LIN {X 0,Y 113.394,Z 388.758,A -85,B 0,C 180,E1 -26470.714,E2 -26470.714} C_VEL
LIN {X 0,Y 109.1,Z 389.64,A -85,B 0,C 180,E1 -26474.93,E2 -26474.93} C_VEL
LIN {X 0,Y 104.868,Z 389.896,A -85,B 0,C 180,E1 -26480.244,E2 -26480.244} C_VEL
LIN {X 0,Y 101.559,Z 389.287,A -85,B 0,C 180,E1 -26485.896,E2 -26485.896} C_VEL
LIN {X 0,Y 99.232,Z 387.805,A -85,B 0,C 180,E1 -26491.803,E2 -26491.803} C_VEL
LIN {X 0,Y 97.668,Z 384.272,A -85,B 0,C 180,E1 -26500.36,E2 -26500.36} C_VEL
LIN {X 0,Y 97.717,Z 379.628,A -85,B 0,C 180,E1 -26507.919,E2 -26507.919} C_VEL
LIN {X 0,Y 98.543,Z 374.936,A -85,B 0,C 180,E1 -26513.645,E2 -26513.645} C_VEL
LIN {X 0,Y 99.92,Z 369.096,A -85,B 0,C 180,E1 -26519.29,E2 -26519.29} C_VEL
LIN {X 0,Y 102.004,Z 361.819,A -85,B 0,C 180,E1 -26524.852,E2 -26524.852} C_VEL
LIN {X 0,Y 104.986,Z 352.316,A -85,B 0,C 180,E1 -26530.446,E2 -26530.446} C_VEL
LIN {X 0,Y 108.19,Z 342.332,A -85,B 0,C 180,E1 -26534.94,E2 -26534.94} C_VEL
LIN {X 0,Y 111.403,Z 331.682,A -85,B 0,C 180,E1 -26538.631,E2 -26538.631} C_VEL
LIN {X 0,Y 114.734,Z 319.038,A -85,B 0,C 180,E1 -26541.907,E2 -26541.907} C_VEL
LIN {X 0,Y 117.58,Z 306.377,A -85,B 0,C 180,E1 -26544.3,E2 -26544.3} C_VEL
LIN {X 0,Y 119.75,Z 292.877,A -85,B 0,C 180,E1 -26546.101,E2 -26546.101} C_VEL
LIN {X 0,Y 121.436,Z 279.148,A -85,B 0,C 180,E1 -26547.229,E2 -26547.229} C_VEL
LIN {X 0,Y 124.892,Z 239.128,A -85,B 0,C 180,E1 -26549.691,E2 -26549.691} C_VEL
LIN {X 0,Y 118.851,Z 223.709,A -85,B 0,C 180,E1 -26552.831,E2 -26552.831} C_VEL
LIN {X 0,Y 112.352,Z 209.651,A -85,B 0,C 180,E1 -26556.477,E2 -26556.477} C_VEL
LIN {X 0,Y 105.334,Z 198.402,A -85,B 0,C 180,E1 -26560.607,E2 -26560.607} C_VEL
LIN {X 0,Y 103.347,Z 195.213,A -85,B 0,C 180,E1 -26561.916,E2 -26561.916} C_VEL
LIN {X 0,Y 101.464,Z 192.565,A -85,B 0,C 180,E1 -26563.185,E2 -26563.185} C_VEL
LIN {X 0,Y 101.019,Z 190.903,A -85,B 0,C 180,E1 -26563.693,E2 -26563.693} C_VEL
LIN {X 0,Y 100.77,Z 190.929,A -85,B 0,C 180,E1 -26570.409,E2 -26570.409} C_VEL
LIN {X 0,Y 100.714,Z 190.936,A -85,B 0,C 180,E1 -26574.889,E2 -26574.889} C_VEL
LIN {X 0,Y 100.681,Z 190.926,A -85,B 0,C 180,E1 -26583.11,E2 -26583.11} C_VEL
LIN {X 0,Y 100.629,Z 190.942,A -85,B 0,C 180,E1 -26589.806,E2 -26589.806} C_VEL
LIN {X 0,Y 100.634,Z 190.932,A -85,B 0,C 180,E1 -26595.706,E2 -26595.706} C_VEL
LIN {X 0,Y 100.619,Z 190.949,A -85,B 0,C 180,E1 -26601.053,E2 -26601.053} C_VEL
LIN {X 0,Y 100.682,Z 190.91,A -85,B 0,C 180,E1 -26606.893,E2 -26606.893} C_VEL
LIN {X 0,Y 100.723,Z 190.936,A -85,B 0,C 180,E1 -26615.252,E2 -26615.252} C_VEL
LIN {X 0,Y 100.77,Z 190.902,A -85,B 0,C 180,E1 -26619.593,E2 -26619.593} C_VEL
LIN {X 0,Y 101.113,Z 190.885,A -85,B 0,C 180,E1 -26627.966,E2 -26627.966} C_VEL
LIN {X 0,Y 101.216,Z 190.86,A -85,B 0,C 180,E1 -26632.019,E2 -26632.019} C_VEL
LIN {X 0,Y 101.822,Z 190.796,A -85,B 0,C 180,E1 -26640.002,E2 -26640.002} C_VEL
LIN {X 0,Y 101.217,Z 190.855,A -85,B 0,C 180,E1 -26647.984,E2 -26647.984} C_VEL
LIN {X 0,Y 101.05,Z 190.897,A -85,B 0,C 180,E1 -26653.17,E2 -26653.17} C_VEL
LIN {X 0,Y 100.772,Z 190.934,A -85,B 0,C 180,E1 -26660.41,E2 -26660.41} C_VEL
LIN {X 0,Y 100.701,Z 190.933,A -85,B 0,C 180,E1 -26664.868,E2 -26664.868} C_VEL
LIN {X 0,Y 100.636,Z 190.954,A -85,B 0,C 180,E1 -26669.698,E2 -26669.698} C_VEL
LIN {X 0,Y 101.603,Z 193.649,A -85,B 0,C 180,E1 -26670.531,E2 -26670.531} C_VEL
LIN {X 0,Y 103.52,Z 196.141,A -85,B 0,C 180,E1 -26671.784,E2 -26671.784} C_VEL
LIN {X 0,Y 109.673,Z 206.47,A -85,B 0,C 180,E1 -26675.645,E2 -26675.645} C_VEL
LIN {X 0,Y 115.294,Z 217.308,A -85,B 0,C 180,E1 -26678.881,E2 -26678.881} C_VEL
LIN {X 0,Y 120.773,Z 232.647,A -85,B 0,C 180,E1 -26682.073,E2 -26682.073} C_VEL
LIN {X 0,Y 124.213,Z 244.441,A -85,B 0,C 180,E1 -26684.089,E2 -26684.089} C_VEL
LIN {X 0,Y 124.314,Z 249.248,A -85,B 0,C 180,E1 -26684.526,E2 -26684.526} C_VEL
LIN {X 0,Y 120.506,Z 292.686,A -85,B 0,C 180,E1 -26687.314,E2 -26687.314} C_VEL
LIN {X 0,Y 118.54,Z 305.908,A -85,B 0,C 180,E1 -26688.732,E2 -26688.732} C_VEL
LIN {X 0,Y 116.204,Z 317.72,A -85,B 0,C 180,E1 -26690.577,E2 -26690.577} C_VEL
LIN {X 0,Y 113.003,Z 330.055,A -85,B 0,C 180,E1 -26693.23,E2 -26693.23} C_VEL
LIN {X 0,Y 109.597,Z 341.808,A -85,B 0,C 180,E1 -26696.664,E2 -26696.664} C_VEL
LIN {X 0,Y 106.566,Z 351.426,A -85,B 0,C 180,E1 -26700.355,E2 -26700.355} C_VEL
LIN {X 0,Y 103.695,Z 360.644,A -85,B 0,C 180,E1 -26704.938,E2 -26704.938} C_VEL
LIN {X 0,Y 101.014,Z 369.603,A -85,B 0,C 180,E1 -26710.702,E2 -26710.702} C_VEL
LIN {X 0,Y 99.294,Z 376.773,A -85,B 0,C 180,E1 -26716.701,E2 -26716.701} C_VEL
LIN {X 0,Y 98.557,Z 381.59,A -85,B 0,C 180,E1 -26721.8,E2 -26721.8} C_VEL
LIN {X 0,Y 98.327,Z 386.191,A -85,B 0,C 180,E1 -26727.951,E2 -26727.951} C_VEL
LIN {X 0,Y 98.286,Z 388.572,A -85,B 0,C 180,E1 -26732.048,E2 -26732.048} C_VEL
LIN {X 0,Y 98.411,Z 391.267,A -85,B 0,C 180,E1 -26738.211,E2 -26738.211} C_VEL
LIN {X 0,Y 100,Z 393.408,A -85,B 0,C 180,E1 -26746.326,E2 -26746.326} C_VEL
LIN {X 0,Y 103.424,Z 394.112,A -85,B 0,C 180,E1 -26754.061,E2 -26754.061} C_VEL
LIN {X 0,Y 108.893,Z 393.383,A -85,B 0,C 180,E1 -26761.085,E2 -26761.085} C_VEL
LIN {X 0,Y 115.931,Z 391.168,A -85,B 0,C 180,E1 -26767.316,E2 -26767.316} C_VEL
LIN {X 0,Y 124.081,Z 387.478,A -85,B 0,C 180,E1 -26772.818,E2 -26772.818} C_VEL
LIN {X 0,Y 131.12,Z 383.572,A -85,B 0,C 180,E1 -26776.351,E2 -26776.351} C_VEL
LIN {X 0,Y 138.522,Z 378.707,A -85,B 0,C 180,E1 -26779.554,E2 -26779.554} C_VEL
LIN {X 0,Y 146.531,Z 372.647,A -85,B 0,C 180,E1 -26782.313,E2 -26782.313} C_VEL
LIN {X 0,Y 154.92,Z 365.206,A -85,B 0,C 180,E1 -26784.742,E2 -26784.742} C_VEL
LIN {X 0,Y 163.564,Z 356.027,A -85,B 0,C 180,E1 -26786.914,E2 -26786.914} C_VEL
LIN {X 0,Y 170.963,Z 346.797,A -85,B 0,C 180,E1 -26788.537,E2 -26788.537} C_VEL
LIN {X 0,Y 178.613,Z 335.405,A -85,B 0,C 180,E1 -26789.955,E2 -26789.955} C_VEL
LIN {X 0,Y 184.843,Z 323.877,A -85,B 0,C 180,E1 -26790.983,E2 -26790.983} C_VEL
LIN {X 0,Y 190.498,Z 310.611,A -85,B 0,C 180,E1 -26791.832,E2 -26791.832} C_VEL
LIN {X 0,Y 194.101,Z 299.386,A -85,B 0,C 180,E1 -26792.328,E2 -26792.328} C_VEL
LIN {X 0,Y 194.458,Z 297.623,A -85,B 0,C 180,E1 -26792.68,E2 -26792.68} C_VEL
LIN {X 0,Y 194.529,Z 296.426,A -85,B 0,C 180,E1 -26793.471,E2 -26793.471} C_VEL
LIN {X 0,Y 194.251,Z 296.2,A -85,B 0,C 180,E1 -26794.794,E2 -26794.794} C_VEL
LIN {X 0,Y 193.484,Z 297.975,A -85,B 0,C 180,E1 -26798.13,E2 -26798.13} C_VEL
LIN {X 0,Y 193.518,Z 298.009,A -85,B 0,C 180,E1 -26798.613,E2 -26798.613} C_VEL
LIN {X 0,Y 193.642,Z 298.314,A -85,B 0,C 180,E1 -26799.96,E2 -26799.96} C_VEL
LIN {X 0,Y 189.131,Z 311.645,A -85,B 0,C 180,E1 -26800.643,E2 -26800.643} C_VEL
LIN {X 0,Y 183.324,Z 324.478,A -85,B 0,C 180,E1 -26801.574,E2 -26801.574} C_VEL
LIN {X 0,Y 176.612,Z 336.059,A -85,B 0,C 180,E1 -26802.751,E2 -26802.751} C_VEL
LIN {X 0,Y 168.731,Z 347.161,A -85,B 0,C 180,E1 -26804.278,E2 -26804.278} C_VEL
LIN {X 0,Y 161.82,Z 355.239,A -85,B 0,C 180,E1 -26805.75,E2 -26805.75} C_VEL
LIN {X 0,Y 153.509,Z 363.475,A -85,B 0,C 180,E1 -26807.76,E2 -26807.76} C_VEL
LIN {X 0,Y 143.868,Z 371.395,A -85,B 0,C 180,E1 -26810.488,E2 -26810.488} C_VEL
LIN {X 0,Y 134.326,Z 377.914,A -85,B 0,C 180,E1 -26813.753,E2 -26813.753} C_VEL
LIN {X 0,Y 126.685,Z 382.18,A -85,B 0,C 180,E1 -26816.91,E2 -26816.91} C_VEL
LIN {X 0,Y 119.479,Z 385.482,A -85,B 0,C 180,E1 -26820.549,E2 -26820.549} C_VEL
LIN {X 0,Y 112.816,Z 387.875,A -85,B 0,C 180,E1 -26824.647,E2 -26824.647} C_VEL
LIN {X 0,Y 106.817,Z 389.413,A -85,B 0,C 180,E1 -26829.287,E2 -26829.287} C_VEL
LIN {X 0,Y 100.124,Z 390.135,A -85,B 0,C 180,E1 -26836.304,E2 -26836.304} C_VEL
LIN {X 0,Y 96.622,Z 389.783,A -85,B 0,C 180,E1 -26841.325,E2 -26841.325} C_VEL
LIN {X 0,Y 93.832,Z 388.808,A -85,B 0,C 180,E1 -26846.703,E2 -26846.703} C_VEL
LIN {X 0,Y 91.202,Z 385.997,A -85,B 0,C 180,E1 -26855.301,E2 -26855.301} C_VEL
LIN {X 0,Y 90.512,Z 383.048,A -85,B 0,C 180,E1 -26861.591,E2 -26861.591} C_VEL
LIN {X 0,Y 90.639,Z 379.163,A -85,B 0,C 180,E1 -26867.946,E2 -26867.946} C_VEL
LIN {X 0,Y 91.636,Z 373.852,A -85,B 0,C 180,E1 -26874.658,E2 -26874.658} C_VEL
LIN {X 0,Y 93.142,Z 367.817,A -85,B 0,C 180,E1 -26880.631,E2 -26880.631} C_VEL
LIN {X 0,Y 95.227,Z 360.904,A -85,B 0,C 180,E1 -26886.053,E2 -26886.053} C_VEL
LIN {X 0,Y 98.32,Z 351.51,A -85,B 0,C 180,E1 -26891.777,E2 -26891.777} C_VEL
LIN {X 0,Y 101.719,Z 341.4,A -85,B 0,C 180,E1 -26896.485,E2 -26896.485} C_VEL
LIN {X 0,Y 105.411,Z 329.532,A -85,B 0,C 180,E1 -26900.608,E2 -26900.608} C_VEL
LIN {X 0,Y 108.633,Z 317.539,A -85,B 0,C 180,E1 -26903.733,E2 -26903.733} C_VEL
LIN {X 0,Y 111.595,Z 304.439,A -85,B 0,C 180,E1 -26906.164,E2 -26906.164} C_VEL
LIN {X 0,Y 113.783,Z 291.045,A -85,B 0,C 180,E1 -26907.922,E2 -26907.922} C_VEL
LIN {X 0,Y 115.568,Z 275.498,A -85,B 0,C 180,E1 -26909.114,E2 -26909.114} C_VEL
LIN {X 0,Y 118.609,Z 240.464,A -85,B 0,C 180,E1 -26911.383,E2 -26911.383} C_VEL
LIN {X 0,Y 113.185,Z 226.664,A -85,B 0,C 180,E1 -26914.475,E2 -26914.475} C_VEL
LIN {X 0,Y 107.453,Z 213.945,A -85,B 0,C 180,E1 -26917.984,E2 -26917.984} C_VEL
LIN {X 0,Y 99.311,Z 200.557,A -85,B 0,C 180,E1 -26923.337,E2 -26923.337} C_VEL
LIN {X 0,Y 97,Z 197.039,A -85,B 0,C 180,E1 -26925.059,E2 -26925.059} C_VEL
LIN {X 0,Y 94.472,Z 194.146,A -85,B 0,C 180,E1 -26926.939,E2 -26926.939} C_VEL
LIN {X 0,Y 93.716,Z 191.812,A -85,B 0,C 180,E1 -26927.879,E2 -26927.879} C_VEL
LIN {X 0,Y 93.628,Z 191.82,A -85,B 0,C 180,E1 -26935.747,E2 -26935.747} C_VEL
LIN {X 0,Y 93.579,Z 191.817,A -85,B 0,C 180,E1 -26944.301,E2 -26944.301} C_VEL
LIN {X 0,Y 93.521,Z 191.808,A -85,B 0,C 180,E1 -26952.558,E2 -26952.558} C_VEL
LIN {X 0,Y 93.527,Z 191.833,A -85,B 0,C 180,E1 -26958.715,E2 -26958.715} C_VEL
LIN {X 0,Y 93.579,Z 191.795,A -85,B 0,C 180,E1 -26965.703,E2 -26965.703} C_VEL
LIN {X 0,Y 93.629,Z 191.822,A -85,B 0,C 180,E1 -26974.256,E2 -26974.256} C_VEL
LIN {X 0,Y 93.64,Z 191.804,A -85,B 0,C 180,E1 -26977.961,E2 -26977.961} C_VEL
LIN {X 0,Y 94.014,Z 191.768,A -85,B 0,C 180,E1 -26987.042,E2 -26987.042} C_VEL
LIN {X 0,Y 94.128,Z 191.746,A -85,B 0,C 180,E1 -26991.414,E2 -26991.414} C_VEL
LIN {X 0,Y 94.751,Z 191.677,A -85,B 0,C 180,E1 -27000.002,E2 -27000.002} C_VEL
LIN {X 0,Y 94.129,Z 191.741,A -85,B 0,C 180,E1 -27008.59,E2 -27008.59} C_VEL
LIN {X 0,Y 93.958,Z 191.779,A -85,B 0,C 180,E1 -27013.495,E2 -27013.495} C_VEL
LIN {X 0,Y 93.635,Z 191.821,A -85,B 0,C 180,E1 -27022.044,E2 -27022.044} C_VEL
LIN {X 0,Y 93.615,Z 191.818,A -85,B 0,C 180,E1 -27025.727,E2 -27025.727} C_VEL
LIN {X 0,Y 94.495,Z 194.57,A -85,B 0,C 180,E1 -27026.654,E2 -27026.654} C_VEL
LIN {X 0,Y 96.723,Z 197.337,A -85,B 0,C 180,E1 -27028.333,E2 -27028.333} C_VEL
LIN {X 0,Y 100.215,Z 202.921,A -85,B 0,C 180,E1 -27030.943,E2 -27030.943} C_VEL
LIN {X 0,Y 105.187,Z 211.401,A -85,B 0,C 180,E1 -27034.281,E2 -27034.281} C_VEL
LIN {X 0,Y 110.057,Z 220.958,A -85,B 0,C 180,E1 -27037.296,E2 -27037.296} C_VEL
LIN {X 0,Y 114.862,Z 234.875,A -85,B 0,C 180,E1 -27040.409,E2 -27040.409} C_VEL
LIN {X 0,Y 118.188,Z 246.008,A -85,B 0,C 180,E1 -27042.492,E2 -27042.492} C_VEL
LIN {X 0,Y 118.164,Z 250.07,A -85,B 0,C 180,E1 -27042.85,E2 -27042.85} C_VEL
LIN {X 0,Y 114.327,Z 291.924,A -85,B 0,C 180,E1 -27045.633,E2 -27045.633} C_VEL
LIN {X 0,Y 112.15,Z 305.956,A -85,B 0,C 180,E1 -27047.193,E2 -27047.193} C_VEL
LIN {X 0,Y 109.847,Z 317.152,A -85,B 0,C 180,E1 -27049.02,E2 -27049.02} C_VEL
LIN {X 0,Y 106.496,Z 329.581,A -85,B 0,C 180,E1 -27051.78,E2 -27051.78} C_VEL
LIN {X 0,Y 103.154,Z 340.625,A -85,B 0,C 180,E1 -27055.122,E2 -27055.122} C_VEL
LIN {X 0,Y 99.746,Z 351.044,A -85,B 0,C 180,E1 -27059.281,E2 -27059.281} C_VEL
LIN {X 0,Y 96.725,Z 360.293,A -85,B 0,C 180,E1 -27064.154,E2 -27064.154} C_VEL
LIN {X 0,Y 94.34,Z 367.912,A -85,B 0,C 180,E1 -27069.276,E2 -27069.276} C_VEL
LIN {X 0,Y 92.395,Z 375.362,A -85,B 0,C 180,E1 -27075.687,E2 -27075.687} C_VEL
LIN {X 0,Y 91.548,Z 380.394,A -85,B 0,C 180,E1 -27081.168,E2 -27081.168} C_VEL
LIN {X 0,Y 91.27,Z 385.199,A -85,B 0,C 180,E1 -27087.793,E2 -27087.793} C_VEL
LIN {X 0,Y 91.254,Z 387.713,A -85,B 0,C 180,E1 -27092.206,E2 -27092.206} C_VEL
LIN {X 0,Y 91.421,Z 390.547,A -85,B 0,C 180,E1 -27098.843,E2 -27098.843} C_VEL
LIN {X 0,Y 93.206,Z 392.966,A -85,B 0,C 180,E1 -27107.553,E2 -27107.553} C_VEL
LIN {X 0,Y 96.974,Z 393.865,A -85,B 0,C 180,E1 -27115.774,E2 -27115.774} C_VEL
LIN {X 0,Y 102.86,Z 393.366,A -85,B 0,C 180,E1 -27123.133,E2 -27123.133} C_VEL
LIN {X 0,Y 110.375,Z 391.434,A -85,B 0,C 180,E1 -27129.548,E2 -27129.548} C_VEL
LIN {X 0,Y 118.992,Z 387.979,A -85,B 0,C 180,E1 -27135.132,E2 -27135.132} C_VEL
LIN {X 0,Y 126.363,Z 384.345,A -85,B 0,C 180,E1 -27138.661,E2 -27138.661} C_VEL
LIN {X 0,Y 134.082,Z 379.734,A -85,B 0,C 180,E1 -27141.833,E2 -27141.833} C_VEL
LIN {X 0,Y 142.358,Z 373.954,A -85,B 0,C 180,E1 -27144.544,E2 -27144.544} C_VEL
LIN {X 0,Y 152.488,Z 365.565,A -85,B 0,C 180,E1 -27147.257,E2 -27147.257} C_VEL
LIN {X 0,Y 161.404,Z 356.639,A -85,B 0,C 180,E1 -27149.311,E2 -27149.311} C_VEL
LIN {X 0,Y 169.808,Z 346.514,A -85,B 0,C 180,E1 -27150.962,E2 -27150.962} C_VEL
LIN {X 0,Y 176.853,Z 336.34,A -85,B 0,C 180,E1 -27152.15,E2 -27152.15} C_VEL
LIN {X 0,Y 183.235,Z 325.172,A -85,B 0,C 180,E1 -27153.093,E2 -27153.093} C_VEL
LIN {X 0,Y 188.695,Z 313.169,A -85,B 0,C 180,E1 -27153.836,E2 -27153.836} C_VEL
LIN {X 0,Y 193.069,Z 300.628,A -85,B 0,C 180,E1 -27154.372,E2 -27154.372} C_VEL
LIN {X 0,Y 193.419,Z 298.769,A -85,B 0,C 180,E1 -27155.436,E2 -27155.436} C_VEL
LIN {X 0,Y 193.437,Z 298.212,A -85,B 0,C 180,E1 -27156.442,E2 -27156.442} C_VEL
LIN {X 0,Y 193.518,Z 298.009,A -85,B 0,C 180,E1 -27158.613,E2 -27158.613} C_VEL
LIN {X 0,Y 193.353,Z 298.825,A -85,B 0,C 180,E1 -27159.078,E2 -27159.078} C_VEL
LIN {X 0,Y 192.714,Z 301.018,A -85,B 0,C 180,E1 -27159.398,E2 -27159.398} C_VEL
LIN {X 0,Y 191.48,Z 304.858,A -85,B 0,C 180,E1 -27159.451,E2 -27159.451} C_VEL
LIN {X 0,Y 187.404,Z 315.101,A -85,B 0,C 180,E1 -27158.818,E2 -27158.818} C_VEL
LIN {X 0,Y 186.095,Z 317.957,A -85,B 0,C 180,E1 -27158.86,E2 -27158.86} C_VEL
LIN {X 0,Y 180.469,Z 328.902,A -85,B 0,C 180,E1 -27159.694,E2 -27159.694} C_VEL
LIN {X 0,Y 173.566,Z 339.73,A -85,B 0,C 180,E1 -27160.8,E2 -27160.8} C_VEL
LIN {X 0,Y 164.884,Z 350.747,A -85,B 0,C 180,E1 -27162.349,E2 -27162.349} C_VEL
LIN {X 0,Y 155.5,Z 360.522,A -85,B 0,C 180,E1 -27164.265,E2 -27164.265} C_VEL
LIN {X 0,Y 145.774,Z 368.828,A -85,B 0,C 180,E1 -27166.585,E2 -27166.585} C_VEL
LIN {X 0,Y 135.827,Z 375.813,A -85,B 0,C 180,E1 -27169.446,E2 -27169.446} C_VEL
LIN {X 0,Y 127.673,Z 380.498,A -85,B 0,C 180,E1 -27172.23,E2 -27172.23} C_VEL
LIN {X 0,Y 117.527,Z 385.189,A -85,B 0,C 180,E1 -27176.57,E2 -27176.57} C_VEL
LIN {X 0,Y 111.089,Z 387.514,A -85,B 0,C 180,E1 -27179.998,E2 -27179.998} C_VEL
LIN {X 0,Y 105.177,Z 389.089,A -85,B 0,C 180,E1 -27183.83,E2 -27183.83} C_VEL
LIN {X 0,Y 99.463,Z 390.084,A -85,B 0,C 180,E1 -27188.426,E2 -27188.426} C_VEL
LIN {X 0,Y 94.146,Z 390.355,A -85,B 0,C 180,E1 -27193.969,E2 -27193.969} C_VEL
LIN {X 0,Y 89.807,Z 389.757,A -85,B 0,C 180,E1 -27200.106,E2 -27200.106} C_VEL
LIN {X 0,Y 86.517,Z 388.308,A -85,B 0,C 180,E1 -27206.68,E2 -27206.68} C_VEL
LIN {X 0,Y 83.976,Z 385.134,A -85,B 0,C 180,E1 -27215.859,E2 -27215.859} C_VEL
LIN {X 0,Y 83.402,Z 381.981,A -85,B 0,C 180,E1 -27222.384,E2 -27222.384} C_VEL
LIN {X 0,Y 83.684,Z 377.846,A -85,B 0,C 180,E1 -27229.096,E2 -27229.096} C_VEL
LIN {X 0,Y 85.04,Z 371.444,A -85,B 0,C 180,E1 -27237.142,E2 -27237.142} C_VEL
LIN {X 0,Y 87.035,Z 364.395,A -85,B 0,C 180,E1 -27243.881,E2 -27243.881} C_VEL
LIN {X 0,Y 89.785,Z 356.227,A -85,B 0,C 180,E1 -27249.931,E2 -27249.931} C_VEL
LIN {X 0,Y 93.309,Z 346.178,A -85,B 0,C 180,E1 -27255.629,E2 -27255.629} C_VEL
LIN {X 0,Y 96.907,Z 335.656,A -85,B 0,C 180,E1 -27260.083,E2 -27260.083} C_VEL
LIN {X 0,Y 100.743,Z 323.192,A -85,B 0,C 180,E1 -27263.994,E2 -27263.994} C_VEL
LIN {X 0,Y 104.002,Z 310.25,A -85,B 0,C 180,E1 -27266.929,E2 -27266.929} C_VEL
LIN {X 0,Y 106.636,Z 297.298,A -85,B 0,C 180,E1 -27268.992,E2 -27268.992} C_VEL
LIN {X 0,Y 108.567,Z 283.803,A -85,B 0,C 180,E1 -27270.396,E2 -27270.396} C_VEL
LIN {X 0,Y 112.543,Z 242.322,A -85,B 0,C 180,E1 -27273.169,E2 -27273.169} C_VEL
LIN {X 0,Y 107.729,Z 229.872,A -85,B 0,C 180,E1 -27276.197,E2 -27276.197} C_VEL
LIN {X 0,Y 102.538,Z 218.119,A -85,B 0,C 180,E1 -27279.647,E2 -27279.647} C_VEL
LIN {X 0,Y 95.323,Z 205.854,A -85,B 0,C 180,E1 -27284.867,E2 -27284.867} C_VEL
LIN {X 0,Y 92.57,Z 201.95,A -85,B 0,C 180,E1 -27287.034,E2 -27287.034} C_VEL
LIN {X 0,Y 90.181,Z 198.633,A -85,B 0,C 180,E1 -27289.076,E2 -27289.076} C_VEL
LIN {X 0,Y 89.56,Z 197.553,A -85,B 0,C 180,E1 -27289.671,E2 -27289.671} C_VEL
LIN {X 0,Y 87.427,Z 195.251,A -85,B 0,C 180,E1 -27291.611,E2 -27291.611} C_VEL
LIN {X 0,Y 86.559,Z 192.704,A -85,B 0,C 180,E1 -27292.843,E2 -27292.843} C_VEL
LIN {X 0,Y 86.45,Z 192.707,A -85,B 0,C 180,E1 -27299.195,E2 -27299.195} C_VEL
LIN {X 0,Y 86.498,Z 192.707,A -85,B 0,C 180,E1 -27305.662,E2 -27305.662} C_VEL
LIN {X 0,Y 86.446,Z 192.688,A -85,B 0,C 180,E1 -27312.974,E2 -27312.974} C_VEL
LIN {X 0,Y 86.45,Z 192.716,A -85,B 0,C 180,E1 -27319.433,E2 -27319.433} C_VEL
LIN {X 0,Y 86.523,Z 192.674,A -85,B 0,C 180,E1 -27325.35,E2 -27325.35} C_VEL
LIN {X 0,Y 86.553,Z 192.703,A -85,B 0,C 180,E1 -27333.276,E2 -27333.276} C_VEL
LIN {X 0,Y 86.589,Z 192.66,A -85,B 0,C 180,E1 -27341.057,E2 -27341.057} C_VEL
LIN {X 0,Y 86.86,Z 192.655,A -85,B 0,C 180,E1 -27346.153,E2 -27346.153} C_VEL
LIN {X 0,Y 87.023,Z 192.635,A -85,B 0,C 180,E1 -27350.707,E2 -27350.707} C_VEL
LIN {X 0,Y 87.681,Z 192.557,A -85,B 0,C 180,E1 -27360.002,E2 -27360.002} C_VEL
LIN {X 0,Y 87.024,Z 192.63,A -85,B 0,C 180,E1 -27369.297,E2 -27369.297} C_VEL
LIN {X 0,Y 86.86,Z 192.66,A -85,B 0,C 180,E1 -27374.05,E2 -27374.05} C_VEL
LIN {X 0,Y 86.566,Z 192.704,A -85,B 0,C 180,E1 -27380.807,E2 -27380.807} C_VEL
LIN {X 0,Y 87.582,Z 195.517,A -85,B 0,C 180,E1 -27382.097,E2 -27382.097} C_VEL
LIN {X 0,Y 89.771,Z 198.091,A -85,B 0,C 180,E1 -27384.091,E2 -27384.091} C_VEL
LIN {X 0,Y 91.803,Z 201.444,A -85,B 0,C 180,E1 -27385.932,E2 -27385.932} C_VEL
LIN {X 0,Y 95.21,Z 206.474,A -85,B 0,C 180,E1 -27388.656,E2 -27388.656} C_VEL
LIN {X 0,Y 100.921,Z 216.687,A -85,B 0,C 180,E1 -27392.94,E2 -27392.94} C_VEL
LIN {X 0,Y 105.009,Z 225.05,A -85,B 0,C 180,E1 -27395.701,E2 -27395.701} C_VEL
LIN {X 0,Y 109.356,Z 237.939,A -85,B 0,C 180,E1 -27398.765,E2 -27398.765} C_VEL
LIN {X 0,Y 112.259,Z 248.266,A -85,B 0,C 180,E1 -27400.821,E2 -27400.821} C_VEL
LIN {X 0,Y 108.112,Z 292.116,A -85,B 0,C 180,E1 -27403.864,E2 -27403.864} C_VEL
LIN {X 0,Y 105.856,Z 305.968,A -85,B 0,C 180,E1 -27405.471,E2 -27405.471} C_VEL
LIN {X 0,Y 103.061,Z 318.595,A -85,B 0,C 180,E1 -27407.67,E2 -27407.67} C_VEL
LIN {X 0,Y 99.596,Z 330.652,A -85,B 0,C 180,E1 -27410.573,E2 -27410.573} C_VEL
LIN {X 0,Y 96.064,Z 341.656,A -85,B 0,C 180,E1 -27414.177,E2 -27414.177} C_VEL
LIN {X 0,Y 92.968,Z 350.658,A -85,B 0,C 180,E1 -27418.05,E2 -27418.05} C_VEL
LIN {X 0,Y 89.802,Z 359.943,A -85,B 0,C 180,E1 -27423.256,E2 -27423.256} C_VEL
LIN {X 0,Y 87.297,Z 367.557,A -85,B 0,C 180,E1 -27428.759,E2 -27428.759} C_VEL
LIN {X 0,Y 85.285,Z 375,A -85,B 0,C 180,E1 -27435.686,E2 -27435.686} C_VEL
LIN {X 0,Y 84.363,Z 380.936,A -85,B 0,C 180,E1 -27442.821,E2 -27442.821} C_VEL
LIN {X 0,Y 84.298,Z 385.547,A -85,B 0,C 180,E1 -27449.999,E2 -27449.999} C_VEL
LIN {X 0,Y 84.218,Z 387.928,A -85,B 0,C 180,E1 -27454.786,E2 -27454.786} C_VEL
LIN {X 0,Y 85.185,Z 391.316,A -85,B 0,C 180,E1 -27464.329,E2 -27464.329} C_VEL
LIN {X 0,Y 88.239,Z 393.191,A -85,B 0,C 180,E1 -27473.467,E2 -27473.467} C_VEL
LIN {X 0,Y 93.603,Z 393.644,A -85,B 0,C 180,E1 -27481.706,E2 -27481.706} C_VEL
LIN {X 0,Y 100.811,Z 392.649,A -85,B 0,C 180,E1 -27488.859,E2 -27488.859} C_VEL
LIN {X 0,Y 109.89,Z 390.092,A -85,B 0,C 180,E1 -27495.289,E2 -27495.289} C_VEL
LIN {X 0,Y 119.156,Z 386.326,A -85,B 0,C 180,E1 -27500.062,E2 -27500.062} C_VEL
LIN {X 0,Y 127.154,Z 382.278,A -85,B 0,C 180,E1 -27503.265,E2 -27503.265} C_VEL
LIN {X 0,Y 135.522,Z 377.237,A -85,B 0,C 180,E1 -27506.07,E2 -27506.07} C_VEL
LIN {X 0,Y 145.831,Z 369.768,A -85,B 0,C 180,E1 -27508.804,E2 -27508.804} C_VEL
LIN {X 0,Y 154.92,Z 361.834,A -85,B 0,C 180,E1 -27510.84,E2 -27510.84} C_VEL
LIN {X 0,Y 162.647,Z 353.849,A -85,B 0,C 180,E1 -27512.349,E2 -27512.349} C_VEL
LIN {X 0,Y 170.557,Z 344.285,A -85,B 0,C 180,E1 -27513.665,E2 -27513.665} C_VEL
LIN {X 0,Y 177.808,Z 333.657,A -85,B 0,C 180,E1 -27514.706,E2 -27514.706} C_VEL
LIN {X 0,Y 184.344,Z 321.867,A -85,B 0,C 180,E1 -27515.533,E2 -27515.533} C_VEL
LIN {X 0,Y 189.618,Z 309.774,A -85,B 0,C 180,E1 -27516.163,E2 -27516.163} C_VEL
LIN {X 0,Y 190.995,Z 305.941,A -85,B 0,C 180,E1 -27516.299,E2 -27516.299} C_VEL
LIN {X 0,Y 191.309,Z 304.957,A -85,B 0,C 180,E1 -27516.692,E2 -27516.692} C_VEL
LIN {X 0,Y 191.329,Z 304.827,A -85,B 0,C 180,E1 -27517.946,E2 -27517.946} C_VEL
LIN {X 0,Y 191.099,Z 305.504,A -85,B 0,C 180,E1 -27518.17,E2 -27518.17} C_VEL
LIN {X 0,Y 186.095,Z 317.957,A -85,B 0,C 180,E1 -27518.86,E2 -27518.86} C_VEL
LIN {X 0,Y 183.51,Z 323.274,A -85,B 0,C 180,E1 -27518.998,E2 -27518.998} C_VEL
LIN {X 0,Y 178.618,Z 331.896,A -85,B 0,C 180,E1 -27518.77,E2 -27518.77} C_VEL
LIN {X 0,Y 173.123,Z 340.058,A -85,B 0,C 180,E1 -27518.643,E2 -27518.643} C_VEL
LIN {X 0,Y 169.599,Z 344.64,A -85,B 0,C 180,E1 -27518.967,E2 -27518.967} C_VEL
LIN {X 0,Y 160.705,Z 354.796,A -85,B 0,C 180,E1 -27520.419,E2 -27520.419} C_VEL
LIN {X 0,Y 152.901,Z 362.231,A -85,B 0,C 180,E1 -27521.893,E2 -27521.893} C_VEL
LIN {X 0,Y 144.328,Z 369.145,A -85,B 0,C 180,E1 -27523.739,E2 -27523.739} C_VEL
LIN {X 0,Y 134.104,Z 376.055,A -85,B 0,C 180,E1 -27526.356,E2 -27526.356} C_VEL
LIN {X 0,Y 126.201,Z 380.423,A -85,B 0,C 180,E1 -27528.76,E2 -27528.76} C_VEL
LIN {X 0,Y 118.307,Z 384.041,A -85,B 0,C 180,E1 -27531.624,E2 -27531.624} C_VEL
LIN {X 0,Y 108.155,Z 387.669,A -85,B 0,C 180,E1 -27536.273,E2 -27536.273} C_VEL
LIN {X 0,Y 98.463,Z 389.882,A -85,B 0,C 180,E1 -27542.216,E2 -27542.216} C_VEL
LIN {X 0,Y 90.6,Z 390.581,A -85,B 0,C 180,E1 -27548.923,E2 -27548.923} C_VEL
LIN {X 0,Y 86.031,Z 390.296,A -85,B 0,C 180,E1 -27554.184,E2 -27554.184} C_VEL
LIN {X 0,Y 82.271,Z 389.364,A -85,B 0,C 180,E1 -27560.008,E2 -27560.008} C_VEL
LIN {X 0,Y 78.126,Z 386.621,A -85,B 0,C 180,E1 -27569.9,E2 -27569.9} C_VEL
LIN {X 0,Y 76.435,Z 382.436,A -85,B 0,C 180,E1 -27580.06,E2 -27580.06} C_VEL
LIN {X 0,Y 76.462,Z 378.455,A -85,B 0,C 180,E1 -27587.331,E2 -27587.331} C_VEL
LIN {X 0,Y 77.43,Z 373.274,A -85,B 0,C 180,E1 -27594.771,E2 -27594.771} C_VEL
LIN {X 0,Y 79.269,Z 366.397,A -85,B 0,C 180,E1 -27602.444,E2 -27602.444} C_VEL
LIN {X 0,Y 82.318,Z 357.585,A -85,B 0,C 180,E1 -27609.901,E2 -27609.901} C_VEL
LIN {X 0,Y 85.72,Z 348.338,A -85,B 0,C 180,E1 -27615.762,E2 -27615.762} C_VEL
LIN {X 0,Y 89.668,Z 337.386,A -85,B 0,C 180,E1 -27620.982,E2 -27620.982} C_VEL
LIN {X 0,Y 93.366,Z 326.337,A -85,B 0,C 180,E1 -27624.843,E2 -27624.843} C_VEL
LIN {X 0,Y 96.948,Z 313.423,A -85,B 0,C 180,E1 -27628.189,E2 -27628.189} C_VEL
LIN {X 0,Y 99.826,Z 301.05,A -85,B 0,C 180,E1 -27630.418,E2 -27630.418} C_VEL
LIN {X 0,Y 102.154,Z 286.915,A -85,B 0,C 180,E1 -27632.142,E2 -27632.142} C_VEL
LIN {X 0,Y 106.585,Z 244.207,A -85,B 0,C 180,E1 -27635.138,E2 -27635.138} C_VEL
LIN {X 0,Y 102.566,Z 233.631,A -85,B 0,C 180,E1 -27637.877,E2 -27637.877} C_VEL
LIN {X 0,Y 97.776,Z 222.365,A -85,B 0,C 180,E1 -27641.437,E2 -27641.437} C_VEL
LIN {X 0,Y 91.116,Z 210.788,A -85,B 0,C 180,E1 -27646.699,E2 -27646.699} C_VEL
LIN {X 0,Y 88.01,Z 206.443,A -85,B 0,C 180,E1 -27649.414,E2 -27649.414} C_VEL
LIN {X 0,Y 85.61,Z 202.878,A -85,B 0,C 180,E1 -27651.793,E2 -27651.793} C_VEL
LIN {X 0,Y 83.475,Z 199.823,A -85,B 0,C 180,E1 -27654.084,E2 -27654.084} C_VEL
LIN {X 0,Y 82.93,Z 198.794,A -85,B 0,C 180,E1 -27654.745,E2 -27654.745} C_VEL
LIN {X 0,Y 80.583,Z 196.616,A -85,B 0,C 180,E1 -27657.337,E2 -27657.337} C_VEL
LIN {X 0,Y 79.537,Z 194.24,A -85,B 0,C 180,E1 -27658.87,E2 -27658.87} C_VEL
LIN {X 0,Y 79.404,Z 193.583,A -85,B 0,C 180,E1 -27659.271,E2 -27659.271} C_VEL
LIN {X 0,Y 79.358,Z 193.597,A -85,B 0,C 180,E1 -27668.311,E2 -27668.311} C_VEL
LIN {X 0,Y 79.348,Z 193.576,A -85,B 0,C 180,E1 -27675.12,E2 -27675.12} C_VEL
LIN {X 0,Y 79.38,Z 193.582,A -85,B 0,C 180,E1 -27682.828,E2 -27682.828} C_VEL
LIN {X 0,Y 79.456,Z 193.583,A -85,B 0,C 180,E1 -27692.192,E2 -27692.192} C_VEL
LIN {X 0,Y 79.467,Z 193.553,A -85,B 0,C 180,E1 -27699.285,E2 -27699.285} C_VEL
LIN {X 0,Y 79.784,Z 193.531,A -85,B 0,C 180,E1 -27705.689,E2 -27705.689} C_VEL
LIN {X 0,Y 79.908,Z 193.524,A -85,B 0,C 180,E1 -27709.871,E2 -27709.871} C_VEL
LIN {X 0,Y 80.61,Z 193.438,A -85,B 0,C 180,E1 -27720.002,E2 -27720.002} C_VEL
LIN {X 0,Y 79.909,Z 193.521,A -85,B 0,C 180,E1 -27730.133,E2 -27730.133} C_VEL
LIN {X 0,Y 79.757,Z 193.652,A -85,B 0,C 180,E1 -27734.74,E2 -27734.74} C_VEL
LIN {X 0,Y 80.527,Z 196.218,A -85,B 0,C 180,E1 -27736.034,E2 -27736.034} C_VEL
LIN {X 0,Y 82.364,Z 198.391,A -85,B 0,C 180,E1 -27738.181,E2 -27738.181} C_VEL
LIN {X 0,Y 83.165,Z 199.15,A -85,B 0,C 180,E1 -27739.053,E2 -27739.053} C_VEL
LIN {X 0,Y 85.159,Z 202.488,A -85,B 0,C 180,E1 -27741.326,E2 -27741.326} C_VEL
LIN {X 0,Y 86.381,Z 204.289,A -85,B 0,C 180,E1 -27742.579,E2 -27742.579} C_VEL
LIN {X 0,Y 90.99,Z 211.356,A -85,B 0,C 180,E1 -27746.814,E2 -27746.814} C_VEL
LIN {X 0,Y 97.032,Z 222.465,A -85,B 0,C 180,E1 -27751.708,E2 -27751.708} C_VEL
LIN {X 0,Y 100.221,Z 229.643,A -85,B 0,C 180,E1 -27754.127,E2 -27754.127} C_VEL
LIN {X 0,Y 104.495,Z 243.091,A -85,B 0,C 180,E1 -27757.443,E2 -27757.443} C_VEL
LIN {X 0,Y 106.31,Z 249.508,A -85,B 0,C 180,E1 -27758.812,E2 -27758.812} C_VEL
LIN {X 0,Y 102.052,Z 292.082,A -85,B 0,C 180,E1 -27761.874,E2 -27761.874} C_VEL
LIN {X 0,Y 99.815,Z 305.188,A -85,B 0,C 180,E1 -27763.439,E2 -27763.439} C_VEL
LIN {X 0,Y 96.873,Z 317.949,A -85,B 0,C 180,E1 -27765.711,E2 -27765.711} C_VEL
LIN {X 0,Y 93.032,Z 330.725,A -85,B 0,C 180,E1 -27768.94,E2 -27768.94} C_VEL
LIN {X 0,Y 89.091,Z 342.308,A -85,B 0,C 180,E1 -27773.022,E2 -27773.022} C_VEL
LIN {X 0,Y 85.519,Z 352.111,A -85,B 0,C 180,E1 -27777.712,E2 -27777.712} C_VEL
LIN {X 0,Y 82.318,Z 361.085,A -85,B 0,C 180,E1 -27783.37,E2 -27783.37} C_VEL
LIN {X 0,Y 79.394,Z 369.805,A -85,B 0,C 180,E1 -27790.612,E2 -27790.612} C_VEL
LIN {X 0,Y 77.77,Z 376.748,A -85,B 0,C 180,E1 -27798.268,E2 -27798.268} C_VEL
LIN {X 0,Y 77.231,Z 381.444,A -85,B 0,C 180,E1 -27804.778,E2 -27804.778} C_VEL
LIN {X 0,Y 77.268,Z 384.507,A -85,B 0,C 180,E1 -27809.999,E2 -27809.999} C_VEL
LIN {X 0,Y 77.262,Z 388.067,A -85,B 0,C 180,E1 -27817.841,E2 -27817.841} C_VEL
LIN {X 0,Y 78.351,Z 390.653,A -85,B 0,C 180,E1 -27825.609,E2 -27825.609} C_VEL
LIN {X 0,Y 81.759,Z 392.733,A -85,B 0,C 180,E1 -27835.454,E2 -27835.454} C_VEL
LIN {X 0,Y 87.639,Z 393.43,A -85,B 0,C 180,E1 -27844.147,E2 -27844.147} C_VEL
LIN {X 0,Y 95.392,Z 392.727,A -85,B 0,C 180,E1 -27851.533,E2 -27851.533} C_VEL
LIN {X 0,Y 104.479,Z 390.564,A -85,B 0,C 180,E1 -27857.724,E2 -27857.724} C_VEL
LIN {X 0,Y 114.759,Z 386.943,A -85,B 0,C 180,E1 -27862.761,E2 -27862.761} C_VEL
LIN {X 0,Y 123.071,Z 383.161,A -85,B 0,C 180,E1 -27865.895,E2 -27865.895} C_VEL
LIN {X 0,Y 131.742,Z 378.379,A -85,B 0,C 180,E1 -27868.597,E2 -27868.597} C_VEL
LIN {X 0,Y 142.354,Z 371.326,A -85,B 0,C 180,E1 -27871.198,E2 -27871.198} C_VEL
LIN {X 0,Y 151.679,Z 363.818,A -85,B 0,C 180,E1 -27873.116,E2 -27873.116} C_VEL
LIN {X 0,Y 161.167,Z 354.631,A -85,B 0,C 180,E1 -27874.8,E2 -27874.8} C_VEL
LIN {X 0,Y 170.084,Z 344.207,A -85,B 0,C 180,E1 -27876.093,E2 -27876.093} C_VEL
LIN {X 0,Y 177.471,Z 333.6,A -85,B 0,C 180,E1 -27877.028,E2 -27877.028} C_VEL
LIN {X 0,Y 178.604,Z 331.729,A -85,B 0,C 180,E1 -27877.63,E2 -27877.63} C_VEL
LIN {X 0,Y 171.611,Z 342.007,A -85,B 0,C 180,E1 -27878.648,E2 -27878.648} C_VEL
LIN {X 0,Y 169.599,Z 344.64,A -85,B 0,C 180,E1 -27878.967,E2 -27878.967} C_VEL
LIN {X 0,Y 165.827,Z 349.181,A -85,B 0,C 180,E1 -27879.331,E2 -27879.331} C_VEL
LIN {X 0,Y 158.982,Z 356.445,A -85,B 0,C 180,E1 -27879.367,E2 -27879.367} C_VEL
LIN {X 0,Y 151.716,Z 363.018,A -85,B 0,C 180,E1 -27879.495,E2 -27879.495} C_VEL
LIN {X 0,Y 147.325,Z 366.551,A -85,B 0,C 180,E1 -27880.043,E2 -27880.043} C_VEL
LIN {X 0,Y 137.314,Z 373.602,A -85,B 0,C 180,E1 -27882.115,E2 -27882.115} C_VEL
LIN {X 0,Y 126.07,Z 379.912,A -85,B 0,C 180,E1 -27884.975,E2 -27884.975} C_VEL
LIN {X 0,Y 114.687,Z 384.932,A -85,B 0,C 180,E1 -27888.652,E2 -27888.652} C_VEL
LIN {X 0,Y 105.688,Z 387.863,A -85,B 0,C 180,E1 -27892.356,E2 -27892.356} C_VEL
LIN {X 0,Y 98.631,Z 389.498,A -85,B 0,C 180,E1 -27895.987,E2 -27895.987} C_VEL
LIN {X 0,Y 91.368,Z 390.555,A -85,B 0,C 180,E1 -27900.684,E2 -27900.684} C_VEL
LIN {X 0,Y 84.832,Z 390.805,A -85,B 0,C 180,E1 -27906.214,E2 -27906.214} C_VEL
LIN {X 0,Y 79.215,Z 390.208,A -85,B 0,C 180,E1 -27912.605,E2 -27912.605} C_VEL
LIN {X 0,Y 73.46,Z 388.08,A -85,B 0,C 180,E1 -27922.497,E2 -27922.497} C_VEL
LIN {X 0,Y 70.223,Z 384.635,A -85,B 0,C 180,E1 -27932.942,E2 -27932.942} C_VEL
LIN {X 0,Y 69.329,Z 381.149,A -85,B 0,C 180,E1 -27940.985,E2 -27940.985} C_VEL
LIN {X 0,Y 69.721,Z 375.536,A -85,B 0,C 180,E1 -27951.019,E2 -27951.019} C_VEL
LIN {X 0,Y 71.125,Z 369.844,A -85,B 0,C 180,E1 -27958.845,E2 -27958.845} C_VEL
LIN {X 0,Y 73.841,Z 361.503,A -85,B 0,C 180,E1 -27967.624,E2 -27967.624} C_VEL
LIN {X 0,Y 76.987,Z 353.239,A -85,B 0,C 180,E1 -27974.107,E2 -27974.107} C_VEL
LIN {X 0,Y 80.846,Z 343.294,A -85,B 0,C 180,E1 -27979.989,E2 -27979.989} C_VEL
LIN {X 0,Y 84.711,Z 332.865,A -85,B 0,C 180,E1 -27984.583,E2 -27984.583} C_VEL
LIN {X 0,Y 88.519,Z 321.361,A -85,B 0,C 180,E1 -27988.295,E2 -27988.295} C_VEL
LIN {X 0,Y 92.127,Z 308.18,A -85,B 0,C 180,E1 -27991.368,E2 -27991.368} C_VEL
LIN {X 0,Y 94.861,Z 295.089,A -85,B 0,C 180,E1 -27993.452,E2 -27993.452} C_VEL
LIN {X 0,Y 96.904,Z 281.053,A -85,B 0,C 180,E1 -27994.865,E2 -27994.865} C_VEL
LIN {X 0,Y 100.654,Z 245.984,A -85,B 0,C 180,E1 -27997.304,E2 -27997.304} C_VEL
LIN {X 0,Y 97.236,Z 236.796,A -85,B 0,C 180,E1 -27999.935,E2 -27999.935} C_VEL
LIN {X 0,Y 93.056,Z 226.51,A -85,B 0,C 180,E1 -28003.423,E2 -28003.423} C_VEL
LIN {X 0,Y 86.908,Z 215.588,A -85,B 0,C 180,E1 -28008.791,E2 -28008.791} C_VEL
LIN {X 0,Y 82.082,Z 208.393,A -85,B 0,C 180,E1 -28013.782,E2 -28013.782} C_VEL
LIN {X 0,Y 79.37,Z 204.498,A -85,B 0,C 180,E1 -28016.988,E2 -28016.988} C_VEL
LIN {X 0,Y 76.855,Z 201.231,A -85,B 0,C 180,E1 -28020.348,E2 -28020.348} C_VEL
LIN {X 0,Y 76.187,Z 199.915,A -85,B 0,C 180,E1 -28021.434,E2 -28021.434} C_VEL
LIN {X 0,Y 73.711,Z 197.939,A -85,B 0,C 180,E1 -28025.185,E2 -28025.185} C_VEL
LIN {X 0,Y 72.562,Z 195.568,A -85,B 0,C 180,E1 -28027.53,E2 -28027.53} C_VEL
LIN {X 0,Y 72.324,Z 194.473,A -85,B 0,C 180,E1 -28028.31,E2 -28028.31} C_VEL
LIN {X 0,Y 72.222,Z 194.476,A -85,B 0,C 180,E1 -28037.068,E2 -28037.068} C_VEL
LIN {X 0,Y 72.282,Z 194.451,A -85,B 0,C 180,E1 -28044.314,E2 -28044.314} C_VEL
LIN {X 0,Y 72.356,Z 194.457,A -85,B 0,C 180,E1 -28050.948,E2 -28050.948} C_VEL
LIN {X 0,Y 72.358,Z 194.456,A -85,B 0,C 180,E1 -28057.141,E2 -28057.141} C_VEL
LIN {X 0,Y 72.676,Z 194.411,A -85,B 0,C 180,E1 -28065.248,E2 -28065.248} C_VEL
LIN {X 0,Y 72.808,Z 194.411,A -85,B 0,C 180,E1 -28068.871,E2 -28068.871} C_VEL
LIN {X 0,Y 73.537,Z 194.318,A -85,B 0,C 180,E1 -28080.002,E2 -28080.002} C_VEL
LIN {X 0,Y 72.932,Z 194.396,A -85,B 0,C 180,E1 -28086.226,E2 -28086.226} C_VEL
LIN {X 0,Y 73.612,Z 196.795,A -85,B 0,C 180,E1 -28087.891,E2 -28087.891} C_VEL
LIN {X 0,Y 75.738,Z 199.332,A -85,B 0,C 180,E1 -28091.383,E2 -28091.383} C_VEL
LIN {X 0,Y 76.605,Z 200.106,A -85,B 0,C 180,E1 -28092.611,E2 -28092.611} C_VEL
LIN {X 0,Y 78.277,Z 203.222,A -85,B 0,C 180,E1 -28095.134,E2 -28095.134} C_VEL
LIN {X 0,Y 80.049,Z 205.338,A -85,B 0,C 180,E1 -28097.32,E2 -28097.32} C_VEL
LIN {X 0,Y 83.046,Z 210.155,A -85,B 0,C 180,E1 -28100.879,E2 -28100.879} C_VEL
LIN {X 0,Y 86.96,Z 216.363,A -85,B 0,C 180,E1 -28104.882,E2 -28104.882} C_VEL
LIN {X 0,Y 92.486,Z 227.008,A -85,B 0,C 180,E1 -28109.818,E2 -28109.818} C_VEL
LIN {X 0,Y 95.095,Z 232.93,A -85,B 0,C 180,E1 -28112.015,E2 -28112.015} C_VEL
LIN {X 0,Y 99.181,Z 246.53,A -85,B 0,C 180,E1 -28115.621,E2 -28115.621} C_VEL
LIN {X 0,Y 100.377,Z 250.951,A -85,B 0,C 180,E1 -28116.64,E2 -28116.64} C_VEL
LIN {X 0,Y 96.117,Z 291.495,A -85,B 0,C 180,E1 -28119.643,E2 -28119.643} C_VEL
LIN {X 0,Y 93.631,Z 305.403,A -85,B 0,C 180,E1 -28121.357,E2 -28121.357} C_VEL
LIN {X 0,Y 90.827,Z 317.05,A -85,B 0,C 180,E1 -28123.496,E2 -28123.496} C_VEL
LIN {X 0,Y 87.079,Z 329.114,A -85,B 0,C 180,E1 -28126.586,E2 -28126.586} C_VEL
LIN {X 0,Y 83.087,Z 340.431,A -85,B 0,C 180,E1 -28130.625,E2 -28130.625} C_VEL
LIN {X 0,Y 79.205,Z 350.58,A -85,B 0,C 180,E1 -28135.551,E2 -28135.551} C_VEL
LIN {X 0,Y 75.428,Z 360.595,A -85,B 0,C 180,E1 -28142.233,E2 -28142.233} C_VEL
LIN {X 0,Y 72.325,Z 369.364,A -85,B 0,C 180,E1 -28150.116,E2 -28150.116} C_VEL
LIN {X 0,Y 70.657,Z 376.347,A -85,B 0,C 180,E1 -28158.525,E2 -28158.525} C_VEL
LIN {X 0,Y 70.186,Z 381.848,A -85,B 0,C 180,E1 -28167.129,E2 -28167.129} C_VEL
LIN {X 0,Y 70.215,Z 384.765,A -85,B 0,C 180,E1 -28172.868,E2 -28172.868} C_VEL
LIN {X 0,Y 70.582,Z 388.156,A -85,B 0,C 180,E1 -28181.486,E2 -28181.486} C_VEL
LIN {X 0,Y 73.197,Z 391.27,A -85,B 0,C 180,E1 -28192.584,E2 -28192.584} C_VEL
LIN {X 0,Y 75.396,Z 392.263,A -85,B 0,C 180,E1 -28197.778,E2 -28197.778} C_VEL
LIN {X 0,Y 81.86,Z 393.177,A -85,B 0,C 180,E1 -28206.938,E2 -28206.938} C_VEL
LIN {X 0,Y 90.206,Z 392.711,A -85,B 0,C 180,E1 -28214.521,E2 -28214.521} C_VEL
LIN {X 0,Y 99.848,Z 390.868,A -85,B 0,C 180,E1 -28220.735,E2 -28220.735} C_VEL
LIN {X 0,Y 105.093,Z 389.396,A -85,B 0,C 180,E1 -28223.366,E2 -28223.366} C_VEL
LIN {X 0,Y 113.508,Z 386.469,A -85,B 0,C 180,E1 -28226.704,E2 -28226.704} C_VEL
LIN {X 0,Y 122.203,Z 382.614,A -85,B 0,C 180,E1 -28229.614,E2 -28229.614} C_VEL
LIN {X 0,Y 131.291,Z 377.766,A -85,B 0,C 180,E1 -28232.033,E2 -28232.033} C_VEL
LIN {X 0,Y 142.294,Z 370.65,A -85,B 0,C 180,E1 -28234.337,E2 -28234.337} C_VEL
LIN {X 0,Y 151.881,Z 363.041,A -85,B 0,C 180,E1 -28236.046,E2 -28236.046} C_VEL
LIN {X 0,Y 159.994,Z 355.405,A -85,B 0,C 180,E1 -28237.285,E2 -28237.285} C_VEL
LIN {X 0,Y 159.18,Z 356.205,A -85,B 0,C 180,E1 -28237.995,E2 -28237.995} C_VEL
LIN {X 0,Y 150.018,Z 364.427,A -85,B 0,C 180,E1 -28239.543,E2 -28239.543} C_VEL
LIN {X 0,Y 147.325,Z 366.551,A -85,B 0,C 180,E1 -28240.043,E2 -28240.043} C_VEL
LIN {X 0,Y 142.736,Z 369.947,A -85,B 0,C 180,E1 -28240.675,E2 -28240.675} C_VEL
LIN {X 0,Y 134.406,Z 375.256,A -85,B 0,C 180,E1 -28241.139,E2 -28241.139} C_VEL
LIN {X 0,Y 125.776,Z 379.868,A -85,B 0,C 180,E1 -28241.746,E2 -28241.746} C_VEL
LIN {X 0,Y 120.764,Z 382.136,A -85,B 0,C 180,E1 -28242.683,E2 -28242.683} C_VEL
LIN {X 0,Y 111.629,Z 385.677,A -85,B 0,C 180,E1 -28245.412,E2 -28245.412} C_VEL
LIN {X 0,Y 99.932,Z 388.971,A -85,B 0,C 180,E1 -28249.918,E2 -28249.918} C_VEL
LIN {X 0,Y 89.376,Z 390.7,A -85,B 0,C 180,E1 -28255.488,E2 -28255.488} C_VEL
LIN {X 0,Y 82.936,Z 391.034,A -85,B 0,C 180,E1 -28259.998,E2 -28259.998} C_VEL
LIN {X 0,Y 77.127,Z 390.783,A -85,B 0,C 180,E1 -28265.226,E2 -28265.226} C_VEL
LIN {X 0,Y 71.779,Z 389.796,A -85,B 0,C 180,E1 -28271.739,E2 -28271.739} C_VEL
LIN {X 0,Y 67.176,Z 387.924,A -85,B 0,C 180,E1 -28279.686,E2 -28279.686} C_VEL
LIN {X 0,Y 64.006,Z 385.202,A -85,B 0,C 180,E1 -28288.552,E2 -28288.552} C_VEL
LIN {X 0,Y 62.317,Z 380.679,A -85,B 0,C 180,E1 -28300.07,E2 -28300.07} C_VEL
LIN {X 0,Y 62.714,Z 374.61,A -85,B 0,C 180,E1 -28311.665,E2 -28311.665} C_VEL
LIN {X 0,Y 64.396,Z 368.276,A -85,B 0,C 180,E1 -28320.815,E2 -28320.815} C_VEL
LIN {X 0,Y 67.353,Z 359.946,A -85,B 0,C 180,E1 -28329.896,E2 -28329.896} C_VEL
LIN {X 0,Y 70.998,Z 350.997,A -85,B 0,C 180,E1 -28337.135,E2 -28337.135} C_VEL
LIN {X 0,Y 75.334,Z 340.488,A -85,B 0,C 180,E1 -28343.304,E2 -28343.304} C_VEL
LIN {X 0,Y 79.679,Z 329.172,A -85,B 0,C 180,E1 -28348.105,E2 -28348.105} C_VEL
LIN {X 0,Y 83.6,Z 317.227,A -85,B 0,C 180,E1 -28351.767,E2 -28351.767} C_VEL
LIN {X 0,Y 87.225,Z 303.725,A -85,B 0,C 180,E1 -28354.622,E2 -28354.622} C_VEL
LIN {X 0,Y 89.793,Z 290.502,A -85,B 0,C 180,E1 -28356.51,E2 -28356.51} C_VEL
LIN {X 0,Y 92.2,Z 271.688,A -85,B 0,C 180,E1 -28358.053,E2 -28358.053} C_VEL
LIN {X 0,Y 94.871,Z 247.696,A -85,B 0,C 180,E1 -28359.752,E2 -28359.752} C_VEL
LIN {X 0,Y 91.865,Z 239.576,A -85,B 0,C 180,E1 -28362.349,E2 -28362.349} C_VEL
LIN {X 0,Y 88.429,Z 230.762,A -85,B 0,C 180,E1 -28365.531,E2 -28365.531} C_VEL
LIN {X 0,Y 83.067,Z 220.685,A -85,B 0,C 180,E1 -28370.852,E2 -28370.852} C_VEL
LIN {X 0,Y 78.346,Z 213.525,A -85,B 0,C 180,E1 -28376.233,E2 -28376.233} C_VEL
LIN {X 0,Y 76.252,Z 210.324,A -85,B 0,C 180,E1 -28379.059,E2 -28379.059} C_VEL
LIN {X 0,Y 73.69,Z 206.507,A -85,B 0,C 180,E1 -28383.053,E2 -28383.053} C_VEL
LIN {X 0,Y 71.012,Z 203.784,A -85,B 0,C 180,E1 -28387.654,E2 -28387.654} C_VEL
LIN {X 0,Y 69.684,Z 201.071,A -85,B 0,C 180,E1 -28390.773,E2 -28390.773} C_VEL
LIN {X 0,Y 66.799,Z 199.079,A -85,B 0,C 180,E1 -28398.12,E2 -28398.12} C_VEL
LIN {X 0,Y 65.155,Z 195.33,A -85,B 0,C 180,E1 -28406.443,E2 -28406.443} C_VEL
LIN {X 0,Y 65.212,Z 195.361,A -85,B 0,C 180,E1 -28414.466,E2 -28414.466} C_VEL
LIN {X 0,Y 65.578,Z 195.287,A -85,B 0,C 180,E1 -28424.693,E2 -28424.693} C_VEL
LIN {X 0,Y 65.774,Z 195.458,A -85,B 0,C 180,E1 -28430.004,E2 -28430.004} C_VEL
LIN {X 0,Y 66.67,Z 197.681,A -85,B 0,C 180,E1 -28434.331,E2 -28434.331} C_VEL
LIN {X 0,Y 70.409,Z 201.116,A -85,B 0,C 180,E1 -28444.029,E2 -28444.029} C_VEL
LIN {X 0,Y 71.839,Z 204.057,A -85,B 0,C 180,E1 -28447.203,E2 -28447.203} C_VEL
LIN {X 0,Y 73.834,Z 206.408,A -85,B 0,C 180,E1 -28450.63,E2 -28450.63} C_VEL
LIN {X 0,Y 76.105,Z 210.078,A -85,B 0,C 180,E1 -28454.224,E2 -28454.224} C_VEL
LIN {X 0,Y 77.524,Z 212.336,A -85,B 0,C 180,E1 -28456.205,E2 -28456.205} C_VEL
LIN {X 0,Y 79.587,Z 215.655,A -85,B 0,C 180,E1 -28458.821,E2 -28458.821} C_VEL
LIN {X 0,Y 83.13,Z 221.598,A -85,B 0,C 180,E1 -28462.876,E2 -28462.876} C_VEL
LIN {X 0,Y 88.213,Z 231.939,A -85,B 0,C 180,E1 -28467.999,E2 -28467.999} C_VEL
LIN {X 0,Y 90.404,Z 237.374,A -85,B 0,C 180,E1 -28470.047,E2 -28470.047} C_VEL
LIN {X 0,Y 94.333,Z 251.358,A -85,B 0,C 180,E1 -28473.951,E2 -28473.951} C_VEL
LIN {X 0,Y 94.518,Z 253.615,A -85,B 0,C 180,E1 -28474.321,E2 -28474.321} C_VEL
LIN {X 0,Y 90.181,Z 292.046,A -85,B 0,C 180,E1 -28477.247,E2 -28477.247} C_VEL
LIN {X 0,Y 87.595,Z 305.627,A -85,B 0,C 180,E1 -28478.99,E2 -28478.99} C_VEL
LIN {X 0,Y 84.347,Z 318.104,A -85,B 0,C 180,E1 -28481.418,E2 -28481.418} C_VEL
LIN {X 0,Y 80.525,Z 329.706,A -85,B 0,C 180,E1 -28484.603,E2 -28484.603} C_VEL
LIN {X 0,Y 76.23,Z 341.027,A -85,B 0,C 180,E1 -28488.937,E2 -28488.937} C_VEL
LIN {X 0,Y 72.184,Z 350.964,A -85,B 0,C 180,E1 -28494.255,E2 -28494.255} C_VEL
LIN {X 0,Y 68.582,Z 360.035,A -85,B 0,C 180,E1 -28500.872,E2 -28500.872} C_VEL
LIN {X 0,Y 65.279,Z 368.818,A -85,B 0,C 180,E1 -28509.518,E2 -28509.518} C_VEL
LIN {X 0,Y 63.552,Z 375.859,A -85,B 0,C 180,E1 -28518.84,E2 -28518.84} C_VEL
LIN {X 0,Y 63.166,Z 380.581,A -85,B 0,C 180,E1 -28526.81,E2 -28526.81} C_VEL
LIN {X 0,Y 63.234,Z 383.666,A -85,B 0,C 180,E1 -28533.185,E2 -28533.185} C_VEL
LIN {X 0,Y 63.691,Z 387.276,A -85,B 0,C 180,E1 -28542.748,E2 -28542.748} C_VEL
LIN {X 0,Y 66.709,Z 390.578,A -85,B 0,C 180,E1 -28554.922,E2 -28554.922} C_VEL
LIN {X 0,Y 72.46,Z 392.458,A -85,B 0,C 180,E1 -28565.586,E2 -28565.586} C_VEL
LIN {X 0,Y 80.55,Z 392.971,A -85,B 0,C 180,E1 -28574.265,E2 -28574.265} C_VEL
LIN {X 0,Y 90.271,Z 392.059,A -85,B 0,C 180,E1 -28581.125,E2 -28581.125} C_VEL
LIN {X 0,Y 101.032,Z 389.767,A -85,B 0,C 180,E1 -28586.587,E2 -28586.587} C_VEL
LIN {X 0,Y 109.791,Z 387.061,A -85,B 0,C 180,E1 -28589.786,E2 -28589.786} C_VEL
LIN {X 0,Y 121.842,Z 382.14,A -85,B 0,C 180,E1 -28593.385,E2 -28593.385} C_VEL
LIN {X 0,Y 131.36,Z 377.206,A -85,B 0,C 180,E1 -28595.437,E2 -28595.437} C_VEL
LIN {X 0,Y 139.66,Z 372.041,A -85,B 0,C 180,E1 -28596.959,E2 -28596.959} C_VEL
LIN {X 0,Y 142.228,Z 370.257,A -85,B 0,C 180,E1 -28597.996,E2 -28597.996} C_VEL
LIN {X 0,Y 132.134,Z 376.542,A -85,B 0,C 180,E1 -28599.957,E2 -28599.957} C_VEL
LIN {X 0,Y 120.764,Z 382.136,A -85,B 0,C 180,E1 -28602.683,E2 -28602.683} C_VEL
LIN {X 0,Y 115.67,Z 384.219,A -85,B 0,C 180,E1 -28603.749,E2 -28603.749} C_VEL
LIN {X 0,Y 106.493,Z 387.218,A -85,B 0,C 180,E1 -28604.939,E2 -28604.939} C_VEL
LIN {X 0,Y 97.257,Z 389.433,A -85,B 0,C 180,E1 -28606.453,E2 -28606.453} C_VEL
LIN {X 0,Y 92.163,Z 390.249,A -85,B 0,C 180,E1 -28608.151,E2 -28608.151} C_VEL
LIN {X 0,Y 85.232,Z 391.05,A -85,B 0,C 180,E1 -28611.672,E2 -28611.672} C_VEL
LIN {X 0,Y 77.426,Z 391.246,A -85,B 0,C 180,E1 -28616.808,E2 -28616.808} C_VEL
LIN {X 0,Y 67.787,Z 390.124,A -85,B 0,C 180,E1 -28625.948,E2 -28625.948} C_VEL
LIN {X 0,Y 62.964,Z 388.636,A -85,B 0,C 180,E1 -28632.896,E2 -28632.896} C_VEL
LIN {X 0,Y 57.634,Z 385.138,A -85,B 0,C 180,E1 -28645.127,E2 -28645.127} C_VEL
LIN {X 0,Y 55.298,Z 379.904,A -85,B 0,C 180,E1 -28659.45,E2 -28659.45} C_VEL
LIN {X 0,Y 55.525,Z 374.542,A -85,B 0,C 180,E1 -28670.74,E2 -28670.74} C_VEL
LIN {X 0,Y 57.146,Z 368.563,A -85,B 0,C 180,E1 -28680.534,E2 -28680.534} C_VEL
LIN {X 0,Y 59.856,Z 360.995,A -85,B 0,C 180,E1 -28689.93,E2 -28689.93} C_VEL
LIN {X 0,Y 63.921,Z 351.624,A -85,B 0,C 180,E1 -28698.452,E2 -28698.452} C_VEL
LIN {X 0,Y 68.388,Z 341.501,A -85,B 0,C 180,E1 -28705.019,E2 -28705.019} C_VEL
LIN {X 0,Y 73.4,Z 329.16,A -85,B 0,C 180,E1 -28710.631,E2 -28710.631} C_VEL
LIN {X 0,Y 77.532,Z 317.337,A -85,B 0,C 180,E1 -28714.383,E2 -28714.383} C_VEL
LIN {X 0,Y 81.125,Z 304.785,A -85,B 0,C 180,E1 -28717.155,E2 -28717.155} C_VEL
LIN {X 0,Y 83.901,Z 291.49,A -85,B 0,C 180,E1 -28719.189,E2 -28719.189} C_VEL
LIN {X 0,Y 86.233,Z 275.505,A -85,B 0,C 180,E1 -28720.537,E2 -28720.537} C_VEL
LIN {X 0,Y 89.18,Z 249.307,A -85,B 0,C 180,E1 -28722.508,E2 -28722.508} C_VEL
LIN {X 0,Y 84.056,Z 235.303,A -85,B 0,C 180,E1 -28727.737,E2 -28727.737} C_VEL
LIN {X 0,Y 79.213,Z 225.721,A -85,B 0,C 180,E1 -28733.161,E2 -28733.161} C_VEL
LIN {X 0,Y 74.714,Z 218.486,A -85,B 0,C 180,E1 -28739.017,E2 -28739.017} C_VEL
LIN {X 0,Y 72.917,Z 215.663,A -85,B 0,C 180,E1 -28741.832,E2 -28741.832} C_VEL
LIN {X 0,Y 70.762,Z 212.378,A -85,B 0,C 180,E1 -28745.656,E2 -28745.656} C_VEL
LIN {X 0,Y 68.337,Z 209.366,A -85,B 0,C 180,E1 -28750.57,E2 -28750.57} C_VEL
LIN {X 0,Y 67.573,Z 207.71,A -85,B 0,C 180,E1 -28752.664,E2 -28752.664} C_VEL
LIN {X 0,Y 64.851,Z 205.284,A -85,B 0,C 180,E1 -28760.96,E2 -28760.96} C_VEL
LIN {X 0,Y 63.771,Z 202.29,A -85,B 0,C 180,E1 -28767.822,E2 -28767.822} C_VEL
LIN {X 0,Y 64.085,Z 202.21,A -85,B 0,C 180,E1 -28787.333,E2 -28787.333} C_VEL
LIN {X 0,Y 64.353,Z 202.714,A -85,B 0,C 180,E1 -28788.978,E2 -28788.978} C_VEL
LIN {X 0,Y 65.766,Z 205.262,A -85,B 0,C 180,E1 -28795.406,E2 -28795.406} C_VEL
LIN {X 0,Y 68.104,Z 207.514,A -85,B 0,C 180,E1 -28801.851,E2 -28801.851} C_VEL
LIN {X 0,Y 69.847,Z 210.793,A -85,B 0,C 180,E1 -28805.968,E2 -28805.968} C_VEL
LIN {X 0,Y 71.138,Z 212.458,A -85,B 0,C 180,E1 -28808.417,E2 -28808.417} C_VEL
LIN {X 0,Y 74.405,Z 218.039,A -85,B 0,C 180,E1 -28814.038,E2 -28814.038} C_VEL
LIN {X 0,Y 77.965,Z 224.166,A -85,B 0,C 180,E1 -28818.929,E2 -28818.929} C_VEL
LIN {X 0,Y 81.351,Z 230.881,A -85,B 0,C 180,E1 -28823.022,E2 -28823.022} C_VEL
LIN {X 0,Y 85.29,Z 240.034,A -85,B 0,C 180,E1 -28827.327,E2 -28827.327} C_VEL
LIN {X 0,Y 89.009,Z 253.972,A -85,B 0,C 180,E1 -28831.519,E2 -28831.519} C_VEL
LIN {X 0,Y 84.616,Z 291.005,A -85,B 0,C 180,E1 -28834.372,E2 -28834.372} C_VEL
LIN {X 0,Y 82.039,Z 304.177,A -85,B 0,C 180,E1 -28836.052,E2 -28836.052} C_VEL
LIN {X 0,Y 78.757,Z 316.608,A -85,B 0,C 180,E1 -28838.456,E2 -28838.456} C_VEL
LIN {X 0,Y 74.431,Z 329.138,A -85,B 0,C 180,E1 -28841.962,E2 -28841.962} C_VEL
LIN {X 0,Y 70.011,Z 340.15,A -85,B 0,C 180,E1 -28846.358,E2 -28846.358} C_VEL
LIN {X 0,Y 65.661,Z 350.235,A -85,B 0,C 180,E1 -28852.015,E2 -28852.015} C_VEL
LIN {X 0,Y 61.769,Z 359.389,A -85,B 0,C 180,E1 -28859.202,E2 -28859.202} C_VEL
LIN {X 0,Y 58.248,Z 368.245,A -85,B 0,C 180,E1 -28868.778,E2 -28868.778} C_VEL
LIN {X 0,Y 56.443,Z 375.362,A -85,B 0,C 180,E1 -28879.235,E2 -28879.235} C_VEL
LIN {X 0,Y 56.184,Z 380.963,A -85,B 0,C 180,E1 -28889.999,E2 -28889.999} C_VEL
LIN {X 0,Y 56.26,Z 383.849,A -85,B 0,C 180,E1 -28897.175,E2 -28897.175} C_VEL
LIN {X 0,Y 56.86,Z 386.253,A -85,B 0,C 180,E1 -28904.311,E2 -28904.311} C_VEL
LIN {X 0,Y 60.359,Z 389.867,A -85,B 0,C 180,E1 -28917.757,E2 -28917.757} C_VEL
LIN {X 0,Y 63.176,Z 391.094,A -85,B 0,C 180,E1 -28923.793,E2 -28923.793} C_VEL
LIN {X 0,Y 71.03,Z 392.523,A -85,B 0,C 180,E1 -28933.835,E2 -28933.835} C_VEL
LIN {X 0,Y 80.683,Z 392.596,A -85,B 0,C 180,E1 -28941.621,E2 -28941.621} C_VEL
LIN {X 0,Y 91.526,Z 391.305,A -85,B 0,C 180,E1 -28947.633,E2 -28947.633} C_VEL
LIN {X 0,Y 103.32,Z 388.578,A -85,B 0,C 180,E1 -28952.16,E2 -28952.16} C_VEL
LIN {X 0,Y 115.736,Z 384.359,A -85,B 0,C 180,E1 -28955.622,E2 -28955.622} C_VEL
LIN {X 0,Y 122.095,Z 381.646,A -85,B 0,C 180,E1 -28957.068,E2 -28957.068} C_VEL
LIN {X 0,Y 124.631,Z 380.392,A -85,B 0,C 180,E1 -28958.117,E2 -28958.117} C_VEL
LIN {X 0,Y 115.238,Z 384.315,A -85,B 0,C 180,E1 -28960.275,E2 -28960.275} C_VEL
LIN {X 0,Y 102.292,Z 388.315,A -85,B 0,C 180,E1 -28964.122,E2 -28964.122} C_VEL
LIN {X 0,Y 92.163,Z 390.249,A -85,B 0,C 180,E1 -28968.151,E2 -28968.151} C_VEL
LIN {X 0,Y 87.122,Z 390.92,A -85,B 0,C 180,E1 -28970.083,E2 -28970.083} C_VEL
LIN {X 0,Y 78.025,Z 391.387,A -85,B 0,C 180,E1 -28972.781,E2 -28972.781} C_VEL
LIN {X 0,Y 69.169,Z 391.06,A -85,B 0,C 180,E1 -28976.206,E2 -28976.206} C_VEL
LIN {X 0,Y 64.684,Z 390.433,A -85,B 0,C 180,E1 -28979.454,E2 -28979.454} C_VEL
LIN {X 0,Y 56.97,Z 388.277,A -85,B 0,C 180,E1 -28989.297,E2 -28989.297} C_VEL
LIN {X 0,Y 52.118,Z 385.535,A -85,B 0,C 180,E1 -28999.282,E2 -28999.282} C_VEL
LIN {X 0,Y 49.1,Z 381.876,A -85,B 0,C 180,E1 -29010.819,E2 -29010.819} C_VEL
LIN {X 0,Y 48.142,Z 377.248,A -85,B 0,C 180,E1 -29023.122,E2 -29023.122} C_VEL
LIN {X 0,Y 48.939,Z 371.702,A -85,B 0,C 180,E1 -29034.942,E2 -29034.942} C_VEL
LIN {X 0,Y 51.074,Z 365.206,A -85,B 0,C 180,E1 -29045.62,E2 -29045.62} C_VEL
LIN {X 0,Y 55.057,Z 356.074,A -85,B 0,C 180,E1 -29056.546,E2 -29056.546} C_VEL
LIN {X 0,Y 59.867,Z 345.98,A -85,B 0,C 180,E1 -29064.887,E2 -29064.887} C_VEL
LIN {X 0,Y 64.525,Z 335.686,A -85,B 0,C 180,E1 -29070.781,E2 -29070.781} C_VEL
LIN {X 0,Y 68.95,Z 324.983,A -85,B 0,C 180,E1 -29075.118,E2 -29075.118} C_VEL
LIN {X 0,Y 73.082,Z 312.87,A -85,B 0,C 180,E1 -29078.643,E2 -29078.643} C_VEL
LIN {X 0,Y 76.675,Z 299.806,A -85,B 0,C 180,E1 -29081.158,E2 -29081.158} C_VEL
LIN {X 0,Y 79.281,Z 286.663,A -85,B 0,C 180,E1 -29082.82,E2 -29082.82} C_VEL
LIN {X 0,Y 83.701,Z 251.058,A -85,B 0,C 180,E1 -29085.549,E2 -29085.549} C_VEL
LIN {X 0,Y 79.571,Z 239.256,A -85,B 0,C 180,E1 -29090.487,E2 -29090.487} C_VEL
LIN {X 0,Y 75.282,Z 230.364,A -85,B 0,C 180,E1 -29095.92,E2 -29095.92} C_VEL
LIN {X 0,Y 70.622,Z 222.168,A -85,B 0,C 180,E1 -29103.299,E2 -29103.299} C_VEL
LIN {X 0,Y 68.087,Z 218.383,A -85,B 0,C 180,E1 -29108.162,E2 -29108.162} C_VEL
LIN {X 0,Y 66,Z 215.286,A -85,B 0,C 180,E1 -29113.241,E2 -29113.241} C_VEL
LIN {X 0,Y 65.415,Z 214.214,A -85,B 0,C 180,E1 -29115.039,E2 -29115.039} C_VEL
LIN {X 0,Y 63.171,Z 211.714,A -85,B 0,C 180,E1 -29123.216,E2 -29123.216} C_VEL
LIN {X 0,Y 62.471,Z 209.26,A -85,B 0,C 180,E1 -29128.975,E2 -29128.975} C_VEL
LIN {X 0,Y 62.488,Z 209.169,A -85,B 0,C 180,E1 -29144.535,E2 -29144.535} C_VEL
LIN {X 0,Y 62.927,Z 209.585,A -85,B 0,C 180,E1 -29147.573,E2 -29147.573} C_VEL
LIN {X 0,Y 64.665,Z 212.491,A -85,B 0,C 180,E1 -29155.718,E2 -29155.718} C_VEL
LIN {X 0,Y 66.003,Z 214.073,A -85,B 0,C 180,E1 -29159.812,E2 -29159.812} C_VEL
LIN {X 0,Y 68.027,Z 217.676,A -85,B 0,C 180,E1 -29165.003,E2 -29165.003} C_VEL
LIN {X 0,Y 71.353,Z 223.61,A -85,B 0,C 180,E1 -29171.589,E2 -29171.589} C_VEL
LIN {X 0,Y 75.592,Z 231.683,A -85,B 0,C 180,E1 -29178.14,E2 -29178.14} C_VEL
LIN {X 0,Y 79.745,Z 241.396,A -85,B 0,C 180,E1 -29183.544,E2 -29183.544} C_VEL
LIN {X 0,Y 81.202,Z 245.859,A -85,B 0,C 180,E1 -29185.408,E2 -29185.408} C_VEL
LIN {X 0,Y 83.488,Z 255.341,A -85,B 0,C 180,E1 -29188.464,E2 -29188.464} C_VEL
LIN {X 0,Y 79.114,Z 290.689,A -85,B 0,C 180,E1 -29191.238,E2 -29191.238} C_VEL
LIN {X 0,Y 76.417,Z 303.908,A -85,B 0,C 180,E1 -29192.943,E2 -29192.943} C_VEL
LIN {X 0,Y 72.808,Z 316.798,A -85,B 0,C 180,E1 -29195.49,E2 -29195.49} C_VEL
LIN {X 0,Y 68.073,Z 329.651,A -85,B 0,C 180,E1 -29199.256,E2 -29199.256} C_VEL
LIN {X 0,Y 63.414,Z 340.544,A -85,B 0,C 180,E1 -29203.914,E2 -29203.914} C_VEL
LIN {X 0,Y 58.368,Z 351.477,A -85,B 0,C 180,E1 -29210.791,E2 -29210.791} C_VEL
LIN {X 0,Y 54.284,Z 360.366,A -85,B 0,C 180,E1 -29218.81,E2 -29218.81} C_VEL
LIN {X 0,Y 50.807,Z 368.983,A -85,B 0,C 180,E1 -29229.767,E2 -29229.767} C_VEL
LIN {X 0,Y 49.237,Z 375.823,A -85,B 0,C 180,E1 -29241.792,E2 -29241.792} C_VEL
LIN {X 0,Y 49.175,Z 379.563,A -85,B 0,C 180,E1 -29249.999,E2 -29249.999} C_VEL
LIN {X 0,Y 49.329,Z 382.659,A -85,B 0,C 180,E1 -29258.189,E2 -29258.189} C_VEL
LIN {X 0,Y 50.768,Z 386.31,A -85,B 0,C 180,E1 -29270.246,E2 -29270.246} C_VEL
LIN {X 0,Y 54.194,Z 389.05,A -85,B 0,C 180,E1 -29281.245,E2 -29281.245} C_VEL
LIN {X 0,Y 57.42,Z 390.406,A -85,B 0,C 180,E1 -29287.731,E2 -29287.731} C_VEL
LIN {X 0,Y 66.097,Z 392.139,A -85,B 0,C 180,E1 -29298.096,E2 -29298.096} C_VEL
LIN {X 0,Y 76.474,Z 392.459,A -85,B 0,C 180,E1 -29305.799,E2 -29305.799} C_VEL
LIN {X 0,Y 87.937,Z 391.434,A -85,B 0,C 180,E1 -29311.534,E2 -29311.534} C_VEL
LIN {X 0,Y 100.213,Z 389.046,A -85,B 0,C 180,E1 -29315.737,E2 -29315.737} C_VEL
LIN {X 0,Y 106.603,Z 387.291,A -85,B 0,C 180,E1 -29317.362,E2 -29317.362} C_VEL
LIN {X 0,Y 107.26,Z 387.041,A -85,B 0,C 180,E1 -29318.277,E2 -29318.277} C_VEL
LIN {X 0,Y 96.389,Z 389.633,A -85,B 0,C 180,E1 -29321.414,E2 -29321.414} C_VEL
LIN {X 0,Y 85.286,Z 391.164,A -85,B 0,C 180,E1 -29325.685,E2 -29325.685} C_VEL
LIN {X 0,Y 77.703,Z 391.494,A -85,B 0,C 180,E1 -29329.576,E2 -29329.576} C_VEL
LIN {X 0,Y 70.629,Z 391.25,A -85,B 0,C 180,E1 -29334.287,E2 -29334.287} C_VEL
LIN {X 0,Y 64.684,Z 390.433,A -85,B 0,C 180,E1 -29339.454,E2 -29339.454} C_VEL
LIN {X 0,Y 60.45,Z 389.65,A -85,B 0,C 180,E1 -29343.157,E2 -29343.157} C_VEL
LIN {X 0,Y 52.797,Z 387.542,A -85,B 0,C 180,E1 -29349.185,E2 -29349.185} C_VEL
LIN {X 0,Y 47.174,Z 385.325,A -85,B 0,C 180,E1 -29355.138,E2 -29355.138} C_VEL
LIN {X 0,Y 44.069,Z 383.369,A -85,B 0,C 180,E1 -29361.02,E2 -29361.02} C_VEL
LIN {X 0,Y 43.391,Z 382.666,A -85,B 0,C 180,E1 -29363.298,E2 -29363.298} C_VEL
LIN {X 0,Y 41.156,Z 377.182,A -85,B 0,C 180,E1 -29380.245,E2 -29380.245} C_VEL
LIN {X 0,Y 41.84,Z 371.209,A -85,B 0,C 180,E1 -29394.957,E2 -29394.957} C_VEL
LIN {X 0,Y 44.414,Z 363.986,A -85,B 0,C 180,E1 -29408.263,E2 -29408.263} C_VEL
LIN {X 0,Y 48.572,Z 355.295,A -85,B 0,C 180,E1 -29419.586,E2 -29419.586} C_VEL
LIN {X 0,Y 53.551,Z 345.6,A -85,B 0,C 180,E1 -29428.121,E2 -29428.121} C_VEL
LIN {X 0,Y 59.271,Z 333.776,A -85,B 0,C 180,E1 -29435.103,E2 -29435.103} C_VEL
LIN {X 0,Y 64.14,Z 322.339,A -85,B 0,C 180,E1 -29439.563,E2 -29439.563} C_VEL
LIN {X 0,Y 68.443,Z 309.999,A -85,B 0,C 180,E1 -29442.889,E2 -29442.889} C_VEL
LIN {X 0,Y 71.649,Z 298.556,A -85,B 0,C 180,E1 -29444.958,E2 -29444.958} C_VEL
LIN {X 0,Y 74.21,Z 285.683,A -85,B 0,C 180,E1 -29446.506,E2 -29446.506} C_VEL
LIN {X 0,Y 78.456,Z 253.923,A -85,B 0,C 180,E1 -29448.84,E2 -29448.84} C_VEL
LIN {X 0,Y 78.197,Z 252.253,A -85,B 0,C 180,E1 -29449.334,E2 -29449.334} C_VEL
LIN {X 0,Y 75.343,Z 243.557,A -85,B 0,C 180,E1 -29453.274,E2 -29453.274} C_VEL
LIN {X 0,Y 71.393,Z 234.687,A -85,B 0,C 180,E1 -29459.229,E2 -29459.229} C_VEL
LIN {X 0,Y 67.502,Z 227.524,A -85,B 0,C 180,E1 -29466.413,E2 -29466.413} C_VEL
LIN {X 0,Y 65.735,Z 224.602,A -85,B 0,C 180,E1 -29470.426,E2 -29470.426} C_VEL
LIN {X 0,Y 63.528,Z 220.808,A -85,B 0,C 180,E1 -29477.088,E2 -29477.088} C_VEL
LIN {X 0,Y 61.484,Z 217.846,A -85,B 0,C 180,E1 -29486.389,E2 -29486.389} C_VEL
LIN {X 0,Y 61.191,Z 216.282,A -85,B 0,C 180,E1 -29490.174,E2 -29490.174} C_VEL
LIN {X 0,Y 61.508,Z 216.262,A -85,B 0,C 180,E1 -29505.702,E2 -29505.702} C_VEL
LIN {X 0,Y 63.2,Z 219.359,A -85,B 0,C 180,E1 -29514.754,E2 -29514.754} C_VEL
LIN {X 0,Y 63.955,Z 220.403,A -85,B 0,C 180,E1 -29517.444,E2 -29517.444} C_VEL
LIN {X 0,Y 66.174,Z 224.91,A -85,B 0,C 180,E1 -29523.999,E2 -29523.999} C_VEL
LIN {X 0,Y 69.035,Z 230.404,A -85,B 0,C 180,E1 -29530.143,E2 -29530.143} C_VEL
LIN {X 0,Y 72.475,Z 237.817,A -85,B 0,C 180,E1 -29536.205,E2 -29536.205} C_VEL
LIN {X 0,Y 76.163,Z 247.484,A -85,B 0,C 180,E1 -29541.663,E2 -29541.663} C_VEL
LIN {X 0,Y 78.282,Z 257.02,A -85,B 0,C 180,E1 -29545.076,E2 -29545.076} C_VEL
LIN {X 0,Y 73.667,Z 291.759,A -85,B 0,C 180,E1 -29547.823,E2 -29547.823} C_VEL
LIN {X 0,Y 70.772,Z 304.732,A -85,B 0,C 180,E1 -29549.521,E2 -29549.521} C_VEL
LIN {X 0,Y 66.995,Z 317.201,A -85,B 0,C 180,E1 -29552.058,E2 -29552.058} C_VEL
LIN {X 0,Y 61.914,Z 330.122,A -85,B 0,C 180,E1 -29556.023,E2 -29556.023} C_VEL
LIN {X 0,Y 56.986,Z 340.851,A -85,B 0,C 180,E1 -29560.94,E2 -29560.94} C_VEL
LIN {X 0,Y 52.05,Z 350.633,A -85,B 0,C 180,E1 -29567.535,E2 -29567.535} C_VEL
LIN {X 0,Y 47.585,Z 359.589,A -85,B 0,C 180,E1 -29576.367,E2 -29576.367} C_VEL
LIN {X 0,Y 43.789,Z 368.293,A -85,B 0,C 180,E1 -29588.83,E2 -29588.83} C_VEL
LIN {X 0,Y 42.178,Z 375.238,A -85,B 0,C 180,E1 -29602.819,E2 -29602.819} C_VEL
LIN {X 0,Y 42.36,Z 380.085,A -85,B 0,C 180,E1 -29615.413,E2 -29615.413} C_VEL
LIN {X 0,Y 43.394,Z 384.069,A -85,B 0,C 180,E1 -29628.898,E2 -29628.898} C_VEL
LIN {X 0,Y 48.284,Z 388.193,A -85,B 0,C 180,E1 -29645.605,E2 -29645.605} C_VEL
LIN {X 0,Y 51.999,Z 389.673,A -85,B 0,C 180,E1 -29652.512,E2 -29652.512} C_VEL
LIN {X 0,Y 61.589,Z 391.65,A -85,B 0,C 180,E1 -29663.011,E2 -29663.011} C_VEL
LIN {X 0,Y 72.719,Z 392.27,A -85,B 0,C 180,E1 -29670.434,E2 -29670.434} C_VEL
LIN {X 0,Y 84.785,Z 391.553,A -85,B 0,C 180,E1 -29675.753,E2 -29675.753} C_VEL
LIN {X 0,Y 91.072,Z 390.665,A -85,B 0,C 180,E1 -29677.821,E2 -29677.821} C_VEL
LIN {X 0,Y 90.743,Z 390.697,A -85,B 0,C 180,E1 -29678.336,E2 -29678.336} C_VEL
LIN {X 0,Y 81.477,Z 391.569,A -85,B 0,C 180,E1 -29681.586,E2 -29681.586} C_VEL
LIN {X 0,Y 68.452,Z 391.471,A -85,B 0,C 180,E1 -29688.148,E2 -29688.148} C_VEL
LIN {X 0,Y 59.608,Z 390.237,A -85,B 0,C 180,E1 -29694.908,E2 -29694.908} C_VEL
LIN {X 0,Y 54.795,Z 389.101,A -85,B 0,C 180,E1 -29699.997,E2 -29699.997} C_VEL
LIN {X 0,Y 46.853,Z 385.64,A -85,B 0,C 180,E1 -29712.999,E2 -29712.999} C_VEL
LIN {X 0,Y 43.391,Z 382.666,A -85,B 0,C 180,E1 -29723.298,E2 -29723.298} C_VEL
LIN {X 0,Y 41.38,Z 380.445,A -85,B 0,C 180,E1 -29730.164,E2 -29730.164} C_VEL
LIN {X 0,Y 39.066,Z 377.867,A -85,B 0,C 180,E1 -29737.04,E2 -29737.04} C_VEL
LIN {X 0,Y 35.546,Z 371.867,A -85,B 0,C 180,E1 -29752.123,E2 -29752.123} C_VEL
LIN {X 0,Y 35.479,Z 368.527,A -85,B 0,C 180,E1 -29760.177,E2 -29760.177} C_VEL
LIN {X 0,Y 35.848,Z 367.371,A -85,B 0,C 180,E1 -29762.762,E2 -29762.762} C_VEL
LIN {X 0,Y 39.513,Z 359.403,A -85,B 0,C 180,E1 -29777.156,E2 -29777.156} C_VEL
LIN {X 0,Y 44.568,Z 350.315,A -85,B 0,C 180,E1 -29787.886,E2 -29787.886} C_VEL
LIN {X 0,Y 49.801,Z 340.802,A -85,B 0,C 180,E1 -29795.299,E2 -29795.299} C_VEL
LIN {X 0,Y 55.009,Z 330.418,A -85,B 0,C 180,E1 -29800.742,E2 -29800.742} C_VEL
LIN {X 0,Y 60.066,Z 318.775,A -85,B 0,C 180,E1 -29804.831,E2 -29804.831} C_VEL
LIN {X 0,Y 64.537,Z 305.785,A -85,B 0,C 180,E1 -29807.836,E2 -29807.836} C_VEL
LIN {X 0,Y 67.961,Z 292.358,A -85,B 0,C 180,E1 -29809.876,E2 -29809.876} C_VEL
LIN {X 0,Y 70.721,Z 275.881,A -85,B 0,C 180,E1 -29811.215,E2 -29811.215} C_VEL
LIN {X 0,Y 73.487,Z 255.278,A -85,B 0,C 180,E1 -29812.717,E2 -29812.717} C_VEL
LIN {X 0,Y 71.322,Z 247.941,A -85,B 0,C 180,E1 -29816.353,E2 -29816.353} C_VEL
LIN {X 0,Y 68.168,Z 240.02,A -85,B 0,C 180,E1 -29822.07,E2 -29822.07} C_VEL
LIN {X 0,Y 64.846,Z 233.289,A -85,B 0,C 180,E1 -29829.181,E2 -29829.181} C_VEL
LIN {X 0,Y 63.379,Z 230.648,A -85,B 0,C 180,E1 -29833.17,E2 -29833.17} C_VEL
LIN {X 0,Y 61.792,Z 227.44,A -85,B 0,C 180,E1 -29838.945,E2 -29838.945} C_VEL
LIN {X 0,Y 60.084,Z 224.464,A -85,B 0,C 180,E1 -29848.422,E2 -29848.422} C_VEL
LIN {X 0,Y 59.906,Z 223.216,A -85,B 0,C 180,E1 -29852.016,E2 -29852.016} C_VEL
LIN {X 0,Y 60.14,Z 223.167,A -85,B 0,C 180,E1 -29863.915,E2 -29863.915} C_VEL
LIN {X 0,Y 62.048,Z 226.749,A -85,B 0,C 180,E1 -29875.01,E2 -29875.01} C_VEL
LIN {X 0,Y 63.863,Z 231.085,A -85,B 0,C 180,E1 -29881.579,E2 -29881.579} C_VEL
LIN {X 0,Y 66.196,Z 236.157,A -85,B 0,C 180,E1 -29887.499,E2 -29887.499} C_VEL
LIN {X 0,Y 69.048,Z 243.031,A -85,B 0,C 180,E1 -29893.382,E2 -29893.382} C_VEL
LIN {X 0,Y 71.903,Z 251.498,A -85,B 0,C 180,E1 -29898.5,E2 -29898.5} C_VEL
LIN {X 0,Y 73.299,Z 258.484,A -85,B 0,C 180,E1 -29901.218,E2 -29901.218} C_VEL
LIN {X 0,Y 68.703,Z 291.29,A -85,B 0,C 180,E1 -29903.765,E2 -29903.765} C_VEL
LIN {X 0,Y 65.599,Z 304.473,A -85,B 0,C 180,E1 -29905.43,E2 -29905.43} C_VEL
LIN {X 0,Y 61.641,Z 316.853,A -85,B 0,C 180,E1 -29907.917,E2 -29907.917} C_VEL
LIN {X 0,Y 56.686,Z 328.838,A -85,B 0,C 180,E1 -29911.528,E2 -29911.528} C_VEL
LIN {X 0,Y 51.36,Z 339.748,A -85,B 0,C 180,E1 -29916.493,E2 -29916.493} C_VEL
LIN {X 0,Y 45.961,Z 349.731,A -85,B 0,C 180,E1 -29923.418,E2 -29923.418} C_VEL
LIN {X 0,Y 40.99,Z 358.793,A -85,B 0,C 180,E1 -29933.122,E2 -29933.122} C_VEL
LIN {X 0,Y 36.778,Z 367.59,A -85,B 0,C 180,E1 -29947.53,E2 -29947.53} C_VEL
LIN {X 0,Y 35.135,Z 374.838,A -85,B 0,C 180,E1 -29964.834,E2 -29964.834} C_VEL
LIN {X 0,Y 35.456,Z 378.956,A -85,B 0,C 180,E1 -29977.625,E2 -29977.625} C_VEL
LIN {X 0,Y 37.924,Z 384.089,A -85,B 0,C 180,E1 -29997.598,E2 -29997.598} C_VEL
LIN {X 0,Y 42.748,Z 387.232,A -85,B 0,C 180,E1 -30011.116,E2 -30011.116} C_VEL
LIN {X 0,Y 47.029,Z 388.871,A -85,B 0,C 180,E1 -30018.346,E2 -30018.346} C_VEL
LIN {X 0,Y 57.603,Z 391.135,A -85,B 0,C 180,E1 -30028.651,E2 -30028.651} C_VEL
LIN {X 0,Y 69.489,Z 392.011,A -85,B 0,C 180,E1 -30035.534,E2 -30035.534} C_VEL
LIN {X 0,Y 75.392,Z 391.961,A -85,B 0,C 180,E1 -30038.104,E2 -30038.104} C_VEL
LIN {X 0,Y 66.492,Z 391.633,A -85,B 0,C 180,E1 -30042.033,E2 -30042.033} C_VEL
LIN {X 0,Y 57.591,Z 390.529,A -85,B 0,C 180,E1 -30047.481,E2 -30047.481} C_VEL
LIN {X 0,Y 49.385,Z 388.575,A -85,B 0,C 180,E1 -30054.957,E2 -30054.957} C_VEL
LIN {X 0,Y 42.339,Z 385.766,A -85,B 0,C 180,E1 -30065.173,E2 -30065.173} C_VEL
LIN {X 0,Y 36.051,Z 380.875,A -85,B 0,C 180,E1 -30082.943,E2 -30082.943} C_VEL
LIN {X 0,Y 34.138,Z 375.4,A -85,B 0,C 180,E1 -30101.528,E2 -30101.528} C_VEL
LIN {X 0,Y 35.415,Z 368.479,A -85,B 0,C 180,E1 -30120.259,E2 -30120.259} C_VEL
LIN {X 0,Y 35.848,Z 367.371,A -85,B 0,C 180,E1 -30122.762,E2 -30122.762} C_VEL
LIN {X 0,Y 36.766,Z 363.817,A -85,B 0,C 180,E1 -30130.055,E2 -30130.055} C_VEL
LIN {X 0,Y 37.117,Z 359.986,A -85,B 0,C 180,E1 -30137.108,E2 -30137.108} C_VEL
LIN {X 0,Y 38.834,Z 350.239,A -85,B 0,C 180,E1 -30152.087,E2 -30152.087} C_VEL
LIN {X 0,Y 41.047,Z 345.721,A -85,B 0,C 180,E1 -30156.696,E2 -30156.696} C_VEL
LIN {X 0,Y 47.455,Z 334.569,A -85,B 0,C 180,E1 -30163.927,E2 -30163.927} C_VEL
LIN {X 0,Y 53.004,Z 323.393,A -85,B 0,C 180,E1 -30168.404,E2 -30168.404} C_VEL
LIN {X 0,Y 58.099,Z 310.516,A -85,B 0,C 180,E1 -30171.799,E2 -30171.799} C_VEL
LIN {X 0,Y 61.892,Z 298.288,A -85,B 0,C 180,E1 -30173.832,E2 -30173.832} C_VEL
LIN {X 0,Y 64.796,Z 284.555,A -85,B 0,C 180,E1 -30175.266,E2 -30175.266} C_VEL
LIN {X 0,Y 68.811,Z 257.238,A -85,B 0,C 180,E1 -30177.07,E2 -30177.07} C_VEL
LIN {X 0,Y 67.39,Z 251.869,A -85,B 0,C 180,E1 -30180.084,E2 -30180.084} C_VEL
LIN {X 0,Y 64.96,Z 245.157,A -85,B 0,C 180,E1 -30185.308,E2 -30185.308} C_VEL
LIN {X 0,Y 62.363,Z 239.108,A -85,B 0,C 180,E1 -30192.137,E2 -30192.137} C_VEL
LIN {X 0,Y 61.121,Z 236.493,A -85,B 0,C 180,E1 -30196.381,E2 -30196.381} C_VEL
LIN {X 0,Y 59.896,Z 233.866,A -85,B 0,C 180,E1 -30201.691,E2 -30201.691} C_VEL
LIN {X 0,Y 58.726,Z 230.445,A -85,B 0,C 180,E1 -30212.174,E2 -30212.174} C_VEL
LIN {X 0,Y 58.639,Z 230.176,A -85,B 0,C 180,E1 -30215.89,E2 -30215.89} C_VEL
LIN {X 0,Y 58.942,Z 230.317,A -85,B 0,C 180,E1 -30223.579,E2 -30223.579} C_VEL
LIN {X 0,Y 60.27,Z 233.345,A -85,B 0,C 180,E1 -30232.779,E2 -30232.779} C_VEL
LIN {X 0,Y 61.691,Z 237.335,A -85,B 0,C 180,E1 -30239.061,E2 -30239.061} C_VEL
LIN {X 0,Y 63.521,Z 242.073,A -85,B 0,C 180,E1 -30244.763,E2 -30244.763} C_VEL
LIN {X 0,Y 65.741,Z 248.053,A -85,B 0,C 180,E1 -30250.146,E2 -30250.146} C_VEL
LIN {X 0,Y 67.858,Z 255.389,A -85,B 0,C 180,E1 -30254.888,E2 -30254.888} C_VEL
LIN {X 0,Y 68.603,Z 259.891,A -85,B 0,C 180,E1 -30256.805,E2 -30256.805} C_VEL
LIN {X 0,Y 64.165,Z 290.387,A -85,B 0,C 180,E1 -30259.059,E2 -30259.059} C_VEL
LIN {X 0,Y 60.774,Z 304.296,A -85,B 0,C 180,E1 -30260.698,E2 -30260.698} C_VEL
LIN {X 0,Y 57.172,Z 315.255,A -85,B 0,C 180,E1 -30262.785,E2 -30262.785} C_VEL
LIN {X 0,Y 51.864,Z 327.537,A -85,B 0,C 180,E1 -30266.135,E2 -30266.135} C_VEL
LIN {X 0,Y 45.437,Z 339.905,A -85,B 0,C 180,E1 -30271.709,E2 -30271.709} C_VEL
LIN {X 0,Y 38.948,Z 350.736,A -85,B 0,C 180,E1 -30279.923,E2 -30279.923} C_VEL
LIN {X 0,Y 33.623,Z 359.557,A -85,B 0,C 180,E1 -30291.164,E2 -30291.164} C_VEL
LIN {X 0,Y 29.31,Z 368.132,A -85,B 0,C 180,E1 -30308.918,E2 -30308.918} C_VEL
LIN {X 0,Y 28.204,Z 374.938,A -85,B 0,C 180,E1 -30329.998,E2 -30329.998} C_VEL
LIN {X 0,Y 28.836,Z 378.53,A -85,B 0,C 180,E1 -30344.104,E2 -30344.104} C_VEL
LIN {X 0,Y 31.898,Z 382.861,A -85,B 0,C 180,E1 -30363.42,E2 -30363.42} C_VEL
LIN {X 0,Y 37.721,Z 386.228,A -85,B 0,C 180,E1 -30378.177,E2 -30378.177} C_VEL
LIN {X 0,Y 48.276,Z 389.411,A -85,B 0,C 180,E1 -30390.861,E2 -30390.861} C_VEL
LIN {X 0,Y 54.256,Z 390.509,A -85,B 0,C 180,E1 -30395.055,E2 -30395.055} C_VEL
LIN {X 0,Y 58.275,Z 391.001,A -85,B 0,C 180,E1 -30398.786,E2 -30398.786} C_VEL
LIN {X 0,Y 46.398,Z 388.527,A -85,B 0,C 180,E1 -30406.864,E2 -30406.864} C_VEL
LIN {X 0,Y 36.129,Z 384.598,A -85,B 0,C 180,E1 -30419.995,E2 -30419.995} C_VEL
LIN {X 0,Y 29.586,Z 379.861,A -85,B 0,C 180,E1 -30438.171,E2 -30438.171} C_VEL
LIN {X 0,Y 27.18,Z 374.584,A -85,B 0,C 180,E1 -30459.135,E2 -30459.135} C_VEL
LIN {X 0,Y 28.155,Z 368.34,A -85,B 0,C 180,E1 -30480.053,E2 -30480.053} C_VEL
LIN {X 0,Y 31.613,Z 361.09,A -85,B 0,C 180,E1 -30497.157,E2 -30497.157} C_VEL
LIN {X 0,Y 36.849,Z 352.525,A -85,B 0,C 180,E1 -30510.002,E2 -30510.002} C_VEL
LIN {X 0,Y 41.047,Z 345.721,A -85,B 0,C 180,E1 -30516.696,E2 -30516.696} C_VEL
LIN {X 0,Y 43.294,Z 341.151,A -85,B 0,C 180,E1 -30520.582,E2 -30520.582} C_VEL
LIN {X 0,Y 45.634,Z 333.152,A -85,B 0,C 180,E1 -30527.466,E2 -30527.466} C_VEL
LIN {X 0,Y 47.995,Z 324.677,A -85,B 0,C 180,E1 -30533.378,E2 -30533.378} C_VEL
LIN {X 0,Y 50.03,Z 319.358,A -85,B 0,C 180,E1 -30535.499,E2 -30535.499} C_VEL
LIN {X 0,Y 54.876,Z 306.971,A -85,B 0,C 180,E1 -30538.067,E2 -30538.067} C_VEL
LIN {X 0,Y 58.741,Z 293.785,A -85,B 0,C 180,E1 -30539.758,E2 -30539.758} C_VEL
LIN {X 0,Y 61.475,Z 279.536,A -85,B 0,C 180,E1 -30540.812,E2 -30540.812} C_VEL
LIN {X 0,Y 64.498,Z 259.066,A -85,B 0,C 180,E1 -30542.115,E2 -30542.115} C_VEL
LIN {X 0,Y 63.437,Z 254.884,A -85,B 0,C 180,E1 -30544.866,E2 -30544.866} C_VEL
LIN {X 0,Y 61.826,Z 249.879,A -85,B 0,C 180,E1 -30549.295,E2 -30549.295} C_VEL
LIN {X 0,Y 59.841,Z 244.274,A -85,B 0,C 180,E1 -30556.258,E2 -30556.258} C_VEL
LIN {X 0,Y 58.284,Z 240.465,A -85,B 0,C 180,E1 -30563.825,E2 -30563.825} C_VEL
LIN {X 0,Y 57.535,Z 237.257,A -85,B 0,C 180,E1 -30573.875,E2 -30573.875} C_VEL
LIN {X 0,Y 57.708,Z 237.371,A -85,B 0,C 180,E1 -30582.726,E2 -30582.726} C_VEL
LIN {X 0,Y 58.549,Z 239.751,A -85,B 0,C 180,E1 -30590.278,E2 -30590.278} C_VEL
LIN {X 0,Y 59.661,Z 243.583,A -85,B 0,C 180,E1 -30596.415,E2 -30596.415} C_VEL
LIN {X 0,Y 61.081,Z 248.179,A -85,B 0,C 180,E1 -30602.043,E2 -30602.043} C_VEL
LIN {X 0,Y 62.589,Z 253.084,A -85,B 0,C 180,E1 -30606.662,E2 -30606.662} C_VEL
LIN {X 0,Y 64.132,Z 259.462,A -85,B 0,C 180,E1 -30610.942,E2 -30610.942} C_VEL
LIN {X 0,Y 64.393,Z 261.428,A -85,B 0,C 180,E1 -30611.846,E2 -30611.846} C_VEL
LIN {X 0,Y 59.894,Z 290.686,A -85,B 0,C 180,E1 -30613.84,E2 -30613.84} C_VEL
LIN {X 0,Y 56.448,Z 304.028,A -85,B 0,C 180,E1 -30615.223,E2 -30615.223} C_VEL
LIN {X 0,Y 52.416,Z 315.53,A -85,B 0,C 180,E1 -30617.19,E2 -30617.19} C_VEL
LIN {X 0,Y 46.812,Z 327.61,A -85,B 0,C 180,E1 -30620.226,E2 -30620.226} C_VEL
LIN {X 0,Y 39.912,Z 339.852,A -85,B 0,C 180,E1 -30625.518,E2 -30625.518} C_VEL
LIN {X 0,Y 33.496,Z 349.659,A -85,B 0,C 180,E1 -30632.936,E2 -30632.936} C_VEL
LIN {X 0,Y 27.375,Z 358.613,A -85,B 0,C 180,E1 -30645.086,E2 -30645.086} C_VEL
LIN {X 0,Y 22.311,Z 367.3,A -85,B 0,C 180,E1 -30666.809,E2 -30666.809} C_VEL
LIN {X 0,Y 21.356,Z 374.23,A -85,B 0,C 180,E1 -30694.721,E2 -30694.721} C_VEL
LIN {X 0,Y 22.194,Z 377.024,A -85,B 0,C 180,E1 -30708.458,E2 -30708.458} C_VEL
LIN {X 0,Y 26.344,Z 381.53,A -85,B 0,C 180,E1 -30731.828,E2 -30731.828} C_VEL
LIN {X 0,Y 33.448,Z 385.092,A -85,B 0,C 180,E1 -30747.185,E2 -30747.185} C_VEL
LIN {X 0,Y 40.726,Z 387.495,A -85,B 0,C 180,E1 -30755.38,E2 -30755.38} C_VEL
LIN {X 0,Y 43.05,Z 388.038,A -85,B 0,C 180,E1 -30758.879,E2 -30758.879} C_VEL
LIN {X 0,Y 33.669,Z 384.785,A -85,B 0,C 180,E1 -30767.947,E2 -30767.947} C_VEL
LIN {X 0,Y 24.178,Z 379.386,A -85,B 0,C 180,E1 -30787.94,E2 -30787.94} C_VEL
LIN {X 0,Y 20.219,Z 373.265,A -85,B 0,C 180,E1 -30817.454,E2 -30817.454} C_VEL
LIN {X 0,Y 21.662,Z 366.458,A -85,B 0,C 180,E1 -30846.088,E2 -30846.088} C_VEL
LIN {X 0,Y 26.167,Z 358.815,A -85,B 0,C 180,E1 -30866.152,E2 -30866.152} C_VEL
LIN {X 0,Y 32.555,Z 349.697,A -85,B 0,C 180,E1 -30879.32,E2 -30879.32} C_VEL
LIN {X 0,Y 38.856,Z 340.182,A -85,B 0,C 180,E1 -30887.094,E2 -30887.094} C_VEL
LIN {X 0,Y 45.205,Z 329.248,A -85,B 0,C 180,E1 -30892.45,E2 -30892.45} C_VEL
LIN {X 0,Y 50.03,Z 319.358,A -85,B 0,C 180,E1 -30895.499,E2 -30895.499} C_VEL
LIN {X 0,Y 51.915,Z 314.016,A -85,B 0,C 180,E1 -30897.308,E2 -30897.308} C_VEL
LIN {X 0,Y 53.624,Z 304.969,A -85,B 0,C 180,E1 -30901.334,E2 -30901.334} C_VEL
LIN {X 0,Y 54.907,Z 295.694,A -85,B 0,C 180,E1 -30904.968,E2 -30904.968} C_VEL
LIN {X 0,Y 55.878,Z 289.937,A -85,B 0,C 180,E1 -30906.165,E2 -30906.165} C_VEL
LIN {X 0,Y 59.649,Z 267.882,A -85,B 0,C 180,E1 -30907.245,E2 -30907.245} C_VEL
LIN {X 0,Y 60.686,Z 261.128,A -85,B 0,C 180,E1 -30907.603,E2 -30907.603} C_VEL
LIN {X 0,Y 59.263,Z 255.426,A -85,B 0,C 180,E1 -30912.734,E2 -30912.734} C_VEL
LIN {X 0,Y 57.785,Z 250.211,A -85,B 0,C 180,E1 -30919.473,E2 -30919.473} C_VEL
LIN {X 0,Y 56.762,Z 247.018,A -85,B 0,C 180,E1 -30926.094,E2 -30926.094} C_VEL
LIN {X 0,Y 56.376,Z 244.197,A -85,B 0,C 180,E1 -30935.647,E2 -30935.647} C_VEL
LIN {X 0,Y 56.489,Z 244.464,A -85,B 0,C 180,E1 -30941.933,E2 -30941.933} C_VEL
LIN {X 0,Y 56.969,Z 246.349,A -85,B 0,C 180,E1 -30947.93,E2 -30947.93} C_VEL
LIN {X 0,Y 57.746,Z 249.855,A -85,B 0,C 180,E1 -30953.631,E2 -30953.631} C_VEL
LIN {X 0,Y 59.103,Z 255.445,A -85,B 0,C 180,E1 -30960.408,E2 -30960.408} C_VEL
LIN {X 0,Y 60.509,Z 262.37,A -85,B 0,C 180,E1 -30965.975,E2 -30965.975} C_VEL
LIN {X 0,Y 60.478,Z 264.018,A -85,B 0,C 180,E1 -30966.467,E2 -30966.467} C_VEL
LIN {X 0,Y 56.151,Z 290.485,A -85,B 0,C 180,E1 -30967.895,E2 -30967.895} C_VEL
LIN {X 0,Y 52.477,Z 304.116,A -85,B 0,C 180,E1 -30968.995,E2 -30968.995} C_VEL
LIN {X 0,Y 48.256,Z 315.518,A -85,B 0,C 180,E1 -30970.555,E2 -30970.555} C_VEL
LIN {X 0,Y 42.382,Z 327.564,A -85,B 0,C 180,E1 -30973.033,E2 -30973.033} C_VEL
LIN {X 0,Y 35.005,Z 339.759,A -85,B 0,C 180,E1 -30977.506,E2 -30977.506} C_VEL
LIN {X 0,Y 27.242,Z 350.516,A -85,B 0,C 180,E1 -30985.448,E2 -30985.448} C_VEL
LIN {X 0,Y 20.361,Z 359.279,A -85,B 0,C 180,E1 -30999.042,E2 -30999.042} C_VEL
LIN {X 0,Y 14.719,Z 368.044,A -85,B 0,C 180,E1 -31030.659,E2 -31030.659} C_VEL
LIN {X 0,Y 14.799,Z 373.421,A -85,B 0,C 180,E1 -31063.731,E2 -31063.731} C_VEL
LIN {X 0,Y 17.091,Z 376.88,A -85,B 0,C 180,E1 -31086.597,E2 -31086.597} C_VEL
LIN {X 0,Y 26.251,Z 382.336,A -85,B 0,C 180,E1 -31113.336,E2 -31113.336} C_VEL
LIN {X 0,Y 27.241,Z 382.748,A -85,B 0,C 180,E1 -31114.792,E2 -31114.792} C_VEL
LIN {X 0,Y 28.721,Z 383.328,A -85,B 0,C 180,E1 -31118.361,E2 -31118.361} C_VEL
LIN {X 0,Y 17.663,Z 377.272,A -85,B 0,C 180,E1 -31139.99,E2 -31139.99} C_VEL
LIN {X 0,Y 13.239,Z 371.144,A -85,B 0,C 180,E1 -31178.311,E2 -31178.311} C_VEL
LIN {X 0,Y 15.652,Z 364.312,A -85,B 0,C 180,E1 -31217.108,E2 -31217.108} C_VEL
LIN {X 0,Y 22.29,Z 355.675,A -85,B 0,C 180,E1 -31240.433,E2 -31240.433} C_VEL
LIN {X 0,Y 29.56,Z 346.41,A -85,B 0,C 180,E1 -31251.286,E2 -31251.286} C_VEL
LIN {X 0,Y 36.284,Z 336.753,A -85,B 0,C 180,E1 -31257.099,E2 -31257.099} C_VEL
LIN {X 0,Y 42.77,Z 325.742,A -85,B 0,C 180,E1 -31260.899,E2 -31260.899} C_VEL
LIN {X 0,Y 48.472,Z 313.566,A -85,B 0,C 180,E1 -31263.559,E2 -31263.559} C_VEL
LIN {X 0,Y 53.455,Z 299.548,A -85,B 0,C 180,E1 -31265.308,E2 -31265.308} C_VEL
LIN {X 0,Y 55.878,Z 289.937,A -85,B 0,C 180,E1 -31266.165,E2 -31266.165} C_VEL
LIN {X 0,Y 56.347,Z 286.081,A -85,B 0,C 180,E1 -31267.06,E2 -31267.06} C_VEL
LIN {X 0,Y 56.083,Z 273.797,A -85,B 0,C 180,E1 -31272.698,E2 -31272.698} C_VEL
LIN {X 0,Y 56.428,Z 269.901,A -85,B 0,C 180,E1 -31273.523,E2 -31273.523} C_VEL
LIN {X 0,Y 57.378,Z 263.597,A -85,B 0,C 180,E1 -31273.904,E2 -31273.904} C_VEL
LIN {X 0,Y 56.672,Z 259.909,A -85,B 0,C 180,E1 -31277.766,E2 -31277.766} C_VEL
LIN {X 0,Y 55.831,Z 255.883,A -85,B 0,C 180,E1 -31283.374,E2 -31283.374} C_VEL
LIN {X 0,Y 55.302,Z 253.552,A -85,B 0,C 180,E1 -31288.756,E2 -31288.756} C_VEL
LIN {X 0,Y 55.232,Z 251.166,A -85,B 0,C 180,E1 -31296.74,E2 -31296.74} C_VEL
LIN {X 0,Y 55.282,Z 251.381,A -85,B 0,C 180,E1 -31300.634,E2 -31300.634} C_VEL
LIN {X 0,Y 55.497,Z 252.973,A -85,B 0,C 180,E1 -31305.534,E2 -31305.534} C_VEL
LIN {X 0,Y 56.195,Z 257.715,A -85,B 0,C 180,E1 -31312.819,E2 -31312.819} C_VEL
LIN {X 0,Y 56.927,Z 262.174,A -85,B 0,C 180,E1 -31317.701,E2 -31317.701} C_VEL
LIN {X 0,Y 57.312,Z 265.12,A -85,B 0,C 180,E1 -31320.145,E2 -31320.145} C_VEL
LIN {X 0,Y 53.158,Z 289.97,A -85,B 0,C 180,E1 -31321.151,E2 -31321.151} C_VEL
LIN {X 0,Y 49.561,Z 303.166,A -85,B 0,C 180,E1 -31321.8,E2 -31321.8} C_VEL
LIN {X 0,Y 44.859,Z 315.528,A -85,B 0,C 180,E1 -31322.836,E2 -31322.836} C_VEL
LIN {X 0,Y 38.763,Z 327.499,A -85,B 0,C 180,E1 -31324.293,E2 -31324.293} C_VEL
LIN {X 0,Y 30.993,Z 339.625,A -85,B 0,C 180,E1 -31327.2,E2 -31327.2} C_VEL
LIN {X 0,Y 23.37,Z 349.356,A -85,B 0,C 180,E1 -31332.202,E2 -31332.202} C_VEL
LIN {X 0,Y 15.296,Z 358.213,A -85,B 0,C 180,E1 -31343.222,E2 -31343.222} C_VEL
LIN {X 0,Y 7.862,Z 366.8,A -85,B 0,C 180,E1 -31383.415,E2 -31383.415} C_VEL
LIN {X 0,Y 8.291,Z 371.584,A -85,B 0,C 180,E1 -31435.744,E2 -31435.744} C_VEL
LIN {X 0,Y 11.257,Z 374.468,A -85,B 0,C 180,E1 -31461.347,E2 -31461.347} C_VEL
LIN {X 0,Y 14.027,Z 376.269,A -85,B 0,C 180,E1 -31477.915,E2 -31477.915} C_VEL
LIN {X 0,Y 6.665,Z 370.278,A -85,B 0,C 180,E1 -31522.32,E2 -31522.32} C_VEL
LIN {X 0,Y 8.969,Z 363.99,A -85,B 0,C 180,E1 -31590.007,E2 -31590.007} C_VEL
LIN {X 0,Y 16.846,Z 355.801,A -85,B 0,C 180,E1 -31614.661,E2 -31614.661} C_VEL
LIN {X 0,Y 25.486,Z 346.02,A -85,B 0,C 180,E1 -31623.474,E2 -31623.474} C_VEL
LIN {X 0,Y 33.193,Z 335.658,A -85,B 0,C 180,E1 -31627.5,E2 -31627.5} C_VEL
LIN {X 0,Y 40.372,Z 323.761,A -85,B 0,C 180,E1 -31629.937,E2 -31629.937} C_VEL
LIN {X 0,Y 46.065,Z 311.597,A -85,B 0,C 180,E1 -31631.526,E2 -31631.526} C_VEL
LIN {X 0,Y 50.719,Z 298.472,A -85,B 0,C 180,E1 -31632.455,E2 -31632.455} C_VEL
LIN {X 0,Y 53.976,Z 284.664,A -85,B 0,C 180,E1 -31633.078,E2 -31633.078} C_VEL
LIN {X 0,Y 56.428,Z 269.901,A -85,B 0,C 180,E1 -31633.523,E2 -31633.523} C_VEL
LIN {X 0,Y 56.389,Z 268.325,A -85,B 0,C 180,E1 -31634.369,E2 -31634.369} C_VEL
LIN {X 0,Y 55.664,Z 266.805,A -85,B 0,C 180,E1 -31637.24,E2 -31637.24} C_VEL
LIN {X 0,Y 54.588,Z 265.199,A -85,B 0,C 180,E1 -31642.013,E2 -31642.013} C_VEL
LIN {X 0,Y 54.484,Z 264.523,A -85,B 0,C 180,E1 -31642.958,E2 -31642.958} C_VEL
LIN {X 0,Y 54.139,Z 261.682,A -85,B 0,C 180,E1 -31647.475,E2 -31647.475} C_VEL
LIN {X 0,Y 53.957,Z 259.861,A -85,B 0,C 180,E1 -31652.198,E2 -31652.198} C_VEL
LIN {X 0,Y 54.043,Z 258.487,A -85,B 0,C 180,E1 -31657.041,E2 -31657.041} C_VEL
LIN {X 0,Y 54.109,Z 258.946,A -85,B 0,C 180,E1 -31661.52,E2 -31661.52} C_VEL
LIN {X 0,Y 54.177,Z 261.251,A -85,B 0,C 180,E1 -31665.795,E2 -31665.795} C_VEL
LIN {X 0,Y 54.583,Z 266.293,A -85,B 0,C 180,E1 -31672.168,E2 -31672.168} C_VEL
LIN {X 0,Y 54.674,Z 267.579,A -85,B 0,C 180,E1 -31673.342,E2 -31673.342} C_VEL
LIN {X 0,Y 50.781,Z 290.049,A -85,B 0,C 180,E1 -31673.767,E2 -31673.767} C_VEL
LIN {X 0,Y 47.269,Z 302.705,A -85,B 0,C 180,E1 -31673.884,E2 -31673.884} C_VEL
LIN {X 0,Y 42.396,Z 315.278,A -85,B 0,C 180,E1 -31674.067,E2 -31674.067} C_VEL
LIN {X 0,Y 36.208,Z 327.198,A -85,B 0,C 180,E1 -31674.146,E2 -31674.146} C_VEL
LIN {X 0,Y 28.246,Z 339.304,A -85,B 0,C 180,E1 -31674.433,E2 -31674.433} C_VEL
LIN {X 0,Y 19.39,Z 350.023,A -85,B 0,C 180,E1 -31675.421,E2 -31675.421} C_VEL
LIN {X 0,Y 10.558,Z 358.7,A -85,B 0,C 180,E1 -31676.966,E2 -31676.966} C_VEL
LIN {X 0,Y 2.704,Z 365.149,A -85,B 0,C 180,E1 -31683.09,E2 -31683.09} C_VEL
LIN {X 0,Y 0.93,Z 366.369,A -85,B 0,C 180,E1 -31680.183,E2 -31680.183} C_VEL
LIN {X 0,Y 9.256,Z 359.59,A -85,B 0,C 180,E1 -31639.408,E2 -31639.408} C_VEL
LIN {X 0,Y 18.615,Z 350.493,A -85,B 0,C 180,E1 -31639.037,E2 -31639.037} C_VEL
LIN {X 0,Y 27.797,Z 339.511,A -85,B 0,C 180,E1 -31639.335,E2 -31639.335} C_VEL
LIN {X 0,Y 35.207,Z 328.378,A -85,B 0,C 180,E1 -31639.673,E2 -31639.673} C_VEL
LIN {X 0,Y 41.744,Z 315.975,A -85,B 0,C 180,E1 -31639.961,E2 -31639.961} C_VEL
LIN {X 0,Y 46.895,Z 303.064,A -85,B 0,C 180,E1 -31640.151,E2 -31640.151} C_VEL
LIN {X 0,Y 50.708,Z 289.377,A -85,B 0,C 180,E1 -31640.385,E2 -31640.385} C_VEL
LIN {X 0,Y 54.744,Z 266.386,A -85,B 0,C 180,E1 -31640.59,E2 -31640.59} C_VEL
LIN {X 0,Y 54.484,Z 264.523,A -85,B 0,C 180,E1 -31642.958,E2 -31642.958} C_VEL
LIN {X 0,Y 54.19,Z 263.898,A -85,B 0,C 180,E1 -31644.927,E2 -31644.927} C_VEL
LIN {X 0,Y 53.472,Z 264.855,A -85,B 0,C 180,E1 -31648.601,E2 -31648.601} C_VEL
LIN {X 0,Y 52.84,Z 266.444,A -85,B 0,C 180,E1 -31653.047,E2 -31653.047} C_VEL
LIN {X 0,Y 52.788,Z 266.373,A -85,B 0,C 180,E1 -31655.155,E2 -31655.155} C_VEL
LIN {X 0,Y 52.9,Z 265.576,A -85,B 0,C 180,E1 -31658.433,E2 -31658.433} C_VEL
LIN {X 0,Y 52.874,Z 266.014,A -85,B 0,C 180,E1 -31659.971,E2 -31659.971} C_VEL
LIN {X 0,Y 52.729,Z 270.232,A -85,B 0,C 180,E1 -31665.98,E2 -31665.98} C_VEL
LIN {X 0,Y 49.3,Z 289.771,A -85,B 0,C 180,E1 -31665.814,E2 -31665.814} C_VEL
LIN {X 0,Y 45.649,Z 302.942,A -85,B 0,C 180,E1 -31665.284,E2 -31665.284} C_VEL
LIN {X 0,Y 41.027,Z 314.914,A -85,B 0,C 180,E1 -31664.489,E2 -31664.489} C_VEL
LIN {X 0,Y 34.936,Z 326.864,A -85,B 0,C 180,E1 -31662.853,E2 -31662.853} C_VEL
LIN {X 0,Y 27.058,Z 339.106,A -85,B 0,C 180,E1 -31659.752,E2 -31659.752} C_VEL
LIN {X 0,Y 22.853,Z 344.636,A -85,B 0,C 180,E1 -31657.315,E2 -31657.315} C_VEL
LIN {X 0,Y 28.36,Z 337.191,A -85,B 0,C 180,E1 -31653.523,E2 -31653.523} C_VEL
LIN {X 0,Y 35.694,Z 325.4,A -85,B 0,C 180,E1 -31650.897,E2 -31650.897} C_VEL
LIN {X 0,Y 41.553,Z 313.397,A -85,B 0,C 180,E1 -31649.514,E2 -31649.514} C_VEL
LIN {X 0,Y 46.702,Z 299.356,A -85,B 0,C 180,E1 -31648.617,E2 -31648.617} C_VEL
LIN {X 0,Y 50.04,Z 285.708,A -85,B 0,C 180,E1 -31648.223,E2 -31648.223} C_VEL
LIN {X 0,Y 52.718,Z 269.967,A -85,B 0,C 180,E1 -31647.933,E2 -31647.933} C_VEL
LIN {X 0,Y 52.758,Z 268.864,A -85,B 0,C 180,E1 -31649.098,E2 -31649.098} C_VEL
LIN {X 0,Y 52.774,Z 266.556,A -85,B 0,C 180,E1 -31654.356,E2 -31654.356} C_VEL
LIN {X 0,Y 52.788,Z 266.373,A -85,B 0,C 180,E1 -31655.155,E2 -31655.155} C_VEL
LIN {X 0,Y 52.739,Z 266.659,A -85,B 0,C 180,E1 -31656.626,E2 -31656.626} C_VEL
LIN {X 0,Y 52.458,Z 268.63,A -85,B 0,C 180,E1 -31658.375,E2 -31658.375} C_VEL
LIN {X 0,Y 51.913,Z 272.226,A -85,B 0,C 180,E1 -31659.373,E2 -31659.373} C_VEL
LIN {X 0,Y 50.518,Z 280.368,A -85,B 0,C 180,E1 -31658.598,E2 -31658.598} C_VEL
LIN {X 0,Y 49.28,Z 287.26,A -85,B 0,C 180,E1 -31657.69,E2 -31657.69} C_VEL
LIN {X 0,Y 47.834,Z 293.788,A -85,B 0,C 180,E1 -31657.236,E2 -31657.236} C_VEL
LIN {X 0,Y 47.781,Z 294.003,A -85,B 0,C 180,E1 -31656.964,E2 -31656.964} C_VEL
LIN {X 0,Y 50.787,Z 278.624,A -85,B 0,C 180,E1 -31656.016,E2 -31656.016} C_VEL
LIN {X 0,Y 51.627,Z 273.465,A -85,B 0,C 180,E1 -31655.9,E2 -31655.9} C_VEL
LIN {X 0,Y 51.655,Z 273.201,A -85,B 0,C 180,E1 -31657.886,E2 -31657.886} C_VEL
LIN {X 0,Y 50.696,Z 279.116,A -85,B 0,C 180,E1 -31658.007,E2 -31658.007} C_VEL
LIN {X 0,Y 49.28,Z 287.26,A -85,B 0,C 180,E1 -31657.69,E2 -31657.69} C_VEL
LIN {X 0,Y 49.245,Z 287.642,A -85,B 0,C 180,E1 -31657.677,E2 -31657.677} C_VEL
LIN {X 0,Y 49.245,Z 600,A -85,B 0,C 180,E1 -31657.677,E2 -31657.677} C_VEL
LIN {X 0,Y 49.245,Z 600,A -85,B 0,C 180,E1 -31657.677,E2 -31657.677}

QRS_NEXT_CUT()

QRS_NEXT()
QRS_HOME()

END
